// TwinCAT 3 PLC project PLC
// ProgramVersion: 3.1.4023.0
// libraries:
//   Tc2_ControllerToolbox, * (Beckhoff Automation GmbH)
//   Tc2_EtherCAT, * (Beckhoff Automation GmbH)
//   Tc2_Math, * (Beckhoff Automation GmbH)
//   Tc2_ModbusRTU, * (Beckhoff Automation GmbH)
//   Tc2_SerialCom, * (Beckhoff Automation GmbH)
//   Tc2_Standard, * (Beckhoff Automation GmbH)
//   Tc2_System, * (Beckhoff Automation GmbH)
//   Tc2_Utilities, * (Beckhoff Automation GmbH)
//   Tc2_XmlDataSrv, * (Beckhoff Automation GmbH)
//   Tc3_EventLogger, * (Beckhoff Automation GmbH)
//   Tc3_Module, * (Beckhoff Automation GmbH)
// project tree:
//   / MAIN.TcPOU, PlcTask.TcTTO, SerialComTask.TcTTO
//   PMShared/Hardware/Common/Enum/CoE/ EBaudrate.TcDUT, EDataFrame.TcDUT
//   PMShared/Hardware/Common/Enum/ DeviceFamily.TcDUT, DeviceLogLevel.TcDUT, SerialFlowControl.TcDUT, SerialParity.TcDUT
//   PMShared/Hardware/Common/ HardwareManager.TcPOU
//   PMShared/Hardware/Common/Struct/Configs/ AppConfig.TcDUT, DeviceConfiguration.TcDUT, SerialCommunication.TcDUT
//   PMShared/Hardware/Common/Struct/Configs/Calibrate/ CalibrateConfig.TcDUT, CalibratePMsConfig.TcDUT, HSPowermeter.TcDUT, HTPowermeter.TcDUT
//   PMShared/Hardware/Common/Struct/Configs/CanOverEthercat/ CanOverEthercat.TcDUT, CanOverEthercatConfig.TcDUT
//   PMShared/Hardware/Common/Struct/Configs/CanOverEthercat/CoEModules/ CoeSerialComSettings.TcDUT
//   PMShared/Hardware/Common/Struct/Configs/CanOverEthercat/CoEModules/SubModules/ BaudRate.TcDUT, DataFrame.TcDUT, EnableRtsCts.TcDUT, EnableXonXoffRx.TcDUT, EnableXonXoffTx.TcDUT, SubIndexModuleBase.TcDUT
//   PMShared/Hardware/Common/Struct/Configs/Devices/Chuck/WaferPresenceSensor/ WaferPresenceSensor.TcDUT
//   PMShared/Hardware/Common/Struct/Configs/Devices/Powermeter/Sensor/ PowermeterSensor.TcDUT
//   PMShared/Hardware/Common/Struct/Configs/Log/ LogConfig.TcDUT
//   PMShared/Hardware/Common/Struct/Configs/NetIdManagement/ NetIdManagement.TcDUT
//   PMShared/Hardware/Common/Struct/Configs/PMs/ LightspeedConfig.TcDUT, PhotoLumConfig.TcDUT, NstConfig.TcDUT, ProcessModulesConfig.TcDUT, PsdConfig.TcDUT
//   PMShared/Hardware/Common/Tools/CoeAccess/ CoeAccess.TcPOU
//   PMShared/Hardware/Common/Tools/PWM/ PwmGenerator.TcPOU
//   PMShared/Hardware/Common/Tools/SerialCommunication/ SerialCom.TcPOU
//   PMShared/Hardware/Devices/AttenuationFilters/ AttenuationFilterBase.TcPOU
//   PMShared/Hardware/Devices/AttenuationFilters/Configs/ AttenuationFilterConfigs.TcDUT, RotatingSwitchConfigs.TcDUT, SliderAttenuationFilterConfigs.TcDUT
//   PMShared/Hardware/Devices/AttenuationFilters/Configs/SerialCommunication/ BkgrdSerialAttenuation.TcPOU, BkgrdSerialSliderAttenuation.TcPOU, BkgrdSerialRotatingSwitch.TcPOU
//   PMShared/Hardware/Devices/AttenuationFilters/Configs/Thorlabs/ELL14K/ EFeedbackMsgAttenuationELL14k.TcDUT, ELL14kAttenuationFilterConfig.TcDUT
//   PMShared/Hardware/Devices/AttenuationFilters/Configs/Thorlabs/ELL18/ EFeedbackMsgAttenuationELL18.TcDUT, ELL18AttenuationFilterConfig.TcDUT
//   PMShared/Hardware/Devices/AttenuationFilters/Configs/Thorlabs/ELL9/ EFeedbackMsgAttenuationELL9.TcDUT, ELL9AttenuationFilterConfig.TcDUT
//   PMShared/Hardware/Devices/AttenuationFilters/Configs/Thorlabs/ELL6/ EFeedbackMsgAttenuationELL6.TcDUT, ELL6AttenuationFilterConfig.TcDUT
//   PMShared/Hardware/Devices/AttenuationFilters/Configs/Thorlabs/FW212C/ EFeedbackMsgAttenuationFW212C.TcDUT, FW212CAttenuationFilterConfig.TcDUT
//   PMShared/Hardware/Devices/AttenuationFilters/Thorlabs/ ELL14KAttenuationFilter.TcPOU, ELL18AttenuationFilter.TcPOU, ELL9AttenuationFilter.TcPOU, ELL6AttenuationFilter.TcPOU, FW212CAttenuationFilter.TcPOU
//   PMShared/Hardware/Devices/Axes/ AxesBase.TcPOU, AxesConst.TcGVL
//   PMShared/Hardware/Devices/Axes/Configs/ AxesConfigs.TcDUT, IoAxisConfig.TcDUT, IoAxisConfig.TcDUT
//   PMShared/Hardware/Devices/Axes/Configs/Owis/ EFeedbackMsgOwisPs10.TcDUT, Ps10OwisAxisConfig.TcDUT
//   PMShared/Hardware/Devices/Axes/Configs/Owis/SerialCommunication/ BkgrdSerialOwisPs10.TcPOU
//   PMShared/Hardware/Devices/Axes/Configs/Stage/ EFeedbackMsgStage.TcDUT, EStagePosition.TcDUT, IoStageAxisConfig.TcDUT, IoStageStruct.TcDUT, EFeedbackMsgStage.TcDUT, EStagePosition.TcDUT, IoStageAxisConfig.TcDUT, IoStageStruct.TcDUT
//   PMShared/Hardware/Devices/Axes/IoAxis/Stage/ IoStageAxis.TcPOU, IoStageAxis.TcPOU
//   PMShared/Hardware/Devices/Axes/Owis/ Ps10Axis.TcPOU
//   PMShared/Hardware/Devices/Chambers/Configs/ EChamberMode.TcDUT, EFeedbackMsgChamberBase.TcDUT, EFeedbackMsgSlitDoor.TcDUT, ESlitDoorPosition.TcDUT, IoChamberBase.TcDUT, ChamberConfigs.TcDUT
//   PMShared/Hardware/Devices/Chambers/Configs/Lightspeed/ IoLightspeed.TcDUT, IoSafetyLS.TcDUT, LightspeedChamberConfig.TcDUT
//   PMShared/Hardware/Devices/Chambers/Configs/PhotoLum/ EFeedbackMsgPhotoLumChamber.TcDUT, IoChamberPhotoLum.TcDUT, PhotoLumChamberConfig.TcDUT
//   PMShared/Hardware/Devices/Chambers/Configs/PSD/ EFeedbackMsgPsdChamber.TcDUT, IoChamberPsd.TcDUT, PsdChamberConfig.TcDUT, SensorId.TcDUT
//   PMShared/Hardware/Devices/Chambers/Lightspeed/ LightspeedChamber.TcPOU
//   PMShared/Hardware/Devices/Chambers/PhotoLum/ PhotoLumChamber.TcPOU
//   PMShared/Hardware/Devices/Chambers/PSD/ PsdChamber.TcPOU
//   PMShared/Hardware/Devices/Chucks/ ChuckBase.TcPOU
//   PMShared/Hardware/Devices/Chucks/Configs/ ChuckConfigs.TcDUT, EFeedbackMsgChuckBase.TcDUT, EMaterialPresence.TcDUT, EWaferSize.TcDUT
//   PMShared/Hardware/Devices/Chucks/Configs/PhotLum/ EFeedbackMsgPhotoLumChuck.TcDUT, IoChuckPhotoLum.TcDUT, PhotoLumChuckConfig.TcDUT
//   PMShared/Hardware/Devices/Chucks/Configs/PSD/ EFeedbackMsgPsdChuck.TcDUT, IoChuckPsd.TcDUT, PsdChuckConfig.TcDUT
//   PMShared/Hardware/Devices/Chucks/PhotoLum/ PhotoLumChuck.TcPOU
//   PMShared/Hardware/Devices/Chucks/PSD/ PsdChuck.TcPOU
//   PMShared/Hardware/Devices/DistanceSensors/Configs/ DistanceSensorConfigs.TcDUT
//   PMShared/Hardware/Devices/DistanceSensors/Configs/MicroEpsilon/ EFeedbackMsgMicroEpsilonDistanceSensor.TcDUT, MicroEpsilonDistanceSensorConfig.TcDUT, IoMicroEpsilonDistanceSensor.TcDUT
//   PMShared/Hardware/Devices/DistanceSensors/ DistanceSensorBase.TcPOU
//   PMShared/Hardware/Devices/DistanceSensors/MicroEpsilon/ MicroEpsilonDistanceSensor.TcPOU
//   PMShared/Hardware/Devices/FastAttenuation/Configs/ FastAttenuationConfigs.TcDUT
//   PMShared/Hardware/Devices/FastAttenuation/Configs/Parallax/ EFeedbackMsgStd900.TcDUT, IoStd900.TcDUT, Std900FastAttenuationConfig.TcDUT
//   PMShared/Hardware/Devices/FastAttenuation/ FastAttenuationBase.TcPOU
//   PMShared/Hardware/Devices/FastAttenuation/Parallax/ Std900FastAttenuation.TcPOU
//   PMShared/Hardware/Devices/Ffus/Astrofan/ Astrofan612Ffu.TcPOU, Constants.TcGVL
//   PMShared/Hardware/Devices/Ffus/Astrofan/Loop/EventRaise/ EventRaised.TcPOU
//   PMShared/Hardware/Devices/Ffus/Astrofan/Loop/FfuSpeedMatrix/ Ffumatrixconfig.TcDUT, FfuSpeed.TcDUT, ScaleSpeed.TcPOU
//   PMShared/Hardware/Devices/Ffus/Configs/Astrofan/ Astrofan612FfuConfig.TcDUT, Astrofan612FfuLoopConfig.TcDUT, Astrofan612FfuEvent.TcDUT, EFeedbackMsgAstrofan612.TcDUT
//   PMShared/Hardware/Devices/Ffus/Configs/ FfuConfigs.TcDUT
//   PMShared/Hardware/Devices/Ffus/ FfuBase.TcPOU
//   PMShared/Hardware/Devices/FiberSwitch/Configs/ FiberSwitchConfigs.TcDUT
//   PMShared/Hardware/Devices/FiberSwitch/Configs/Leoni/ EFeedbackMsgEol.TcDUT, EOLFiberSwitchConfig.TcDUT
//   PMShared/Hardware/Devices/FiberSwitch/Configs/SerialCommunication/ BkgrdSerialFiberSwitch.TcPOU
//   PMShared/Hardware/Devices/FiberSwitch/ FiberSwitchBase.TcPOU
//   PMShared/Hardware/Devices/FiberSwitch/Leoni/ EOLFiberSwitch.TcPOU
//   PMShared/Hardware/Devices/Ionizers/Configs/ IonizerAlarm.TcDUT, IonizerConfigs.TcDUT, IonizerConst.TcGVL
//   PMShared/Hardware/Devices/Ionizers/Configs/Keyence/ EFeedbackMsgSJH108.TcDUT, IoSJH108A.TcDUT, SJH108IonizerConfig.TcDUT
//   PMShared/Hardware/Devices/Ionizers/ IonizerBase.TcPOU
//   PMShared/Hardware/Devices/Ionizers/Keyence/ SJH108Ionizer.TcPOU
//   PMShared/Hardware/Devices/Lasers/Coherent/ Sapphire488Laser.TcPOU
//   PMShared/Hardware/Devices/Lasers/Configs/Base/ HoursStruct.TcDUT
//   PMShared/Hardware/Devices/Lasers/Configs/Coherent/ EFeedbackMsgSapphire488.TcDUT, Sapphire488LaserConfig.TcDUT
//   PMShared/Hardware/Devices/Lasers/Configs/ LaserConfigs.TcDUT
//   PMShared/Hardware/Devices/Lasers/Configs/Leukos/ EControlModePiano450.TcDUT, EFeedbackMsgPiano450.TcDUT, Piano450LaserConfig.TcDUT
//   PMShared/Hardware/Devices/Lasers/Configs/Quantum/ EControlModeSmd12.TcDUT, EFeedbackMsgSMD12.TcDUT, SMD12LaserConfig.TcDUT
//   PMShared/Hardware/Devices/Lasers/Configs/SerialCommunication/ BkgrdSerialLaser.TcPOU
//   PMShared/Hardware/Devices/Lasers/ LaserBase.TcPOU
//   PMShared/Hardware/Devices/Lasers/Leukos/ Piano450Laser.TcPOU
//   PMShared/Hardware/Devices/Lasers/Quantum/ SMD12Laser.TcPOU
//   PMShared/Hardware/Devices/Lights/Arduino/ ArduinoLight.TcPOU
//   PMShared/Hardware/Devices/Lights/Configs/Evosens/ EvosensLightConfig.TcDUT, EFeedbackMsgEvosensLight.TcDUT
//   PMShared/Hardware/Devices/Lights/Configs/Arduino/ EFeedbackMsgArduinoLight.TcDUT, ArduinoLightConfig.TcDUT
//   PMShared/Hardware/Devices/Lights/Configs/ LightConfigs.TcDUT
//   PMShared/Hardware/Devices/Lights/Configs/SerialCommunication/ BkgrdSerialLight.TcPOU
//   PMShared/Hardware/Devices/Lights/Evosens/ EvosensLight.TcPOU
//   PMShared/Hardware/Devices/Lights/ LightBase.TcPOU
//   PMShared/Hardware/Devices/MPPCs/Configs/Hamamatsu/ C13336MppcConfig.TcDUT, EFeedbackMsgC13336.TcDUT, EMppcCollector.TcDUT, EMppcStateModule.TcDUT, IoC13336Mppc.TcDUT
//   PMShared/Hardware/Devices/MPPCs/Configs/ MppcConfigs.TcDUT
//   PMShared/Hardware/Devices/MPPCs/Configs/SerialCommunication/ BkgrdSerialMppcNarrow.TcPOU, BkgrdSerialMppcWide.TcPOU
//   PMShared/Hardware/Devices/MPPCs/Hamamatsu/C13336/ C13336MppcWide.TcPOU, C13366MppcNarrow.TcPOU
//   PMShared/Hardware/Devices/MPPCs/Hamamatsu/ C13336Mppc.TcPOU
//   PMShared/Hardware/Devices/MPPCs/ MppcBase.TcPOU
//   PMShared/Hardware/Devices/OpticalPowermeters/Configs/ OpticalPowermeterConfigs.TcDUT
//   PMShared/Hardware/Devices/OpticalPowermeters/Configs/SerialCommunication/ BkgrdSerialOpticalPowermeterHs.TcPOU, BkgrdSerialOpticalPowermeterHt.TcPOU
//   PMShared/Hardware/Devices/OpticalPowermeters/Configs/Thorlabs/ EFeedbackMsgPM101.TcDUT, EPowerIlluminationFlow.TcDUT, IoControlPM101.TcDUT, PM101OpticalPowermeterConfig.TcDUT
//   PMShared/Hardware/Devices/OpticalPowermeters/ OpticalPowermeterBase.TcPOU
//   PMShared/Hardware/Devices/OpticalPowermeters/Thorlabs/PM101/Messages/ BeamDiameterMsg.TcDUT, AttenuationMsg.TcDUT, SensorTypeMsg.TcDUT, ResponsivityMsg.TcDUT, CustomMsg.TcDUT, IdentifierMsg.TcDUT, MaxPowerMsg.TcDUT, MinPowerMsg.TcDUT, PowerMsg.TcDUT, WavelengthMsg.TcDUT, WavelengthRangeMsg.TcDUT
//   PMShared/Hardware/Devices/OpticalPowermeters/Thorlabs/PM101/ PM101OpticalPowermeterHs.TcPOU, PM101OpticalPowermeterHt.TcPOU
//   PMShared/Hardware/Devices/OpticalPowermeters/Thorlabs/ PM101OpticalPowermeter.TcPOU
//   PMShared/Hardware/Devices/PolarisationFilters/Configs/ PolarisationFilterConfigs.TcDUT
//   PMShared/Hardware/Devices/PolarisationFilters/Configs/SerialCommunication/ BkgrdSerialPolarisation.TcPOU
//   PMShared/Hardware/Devices/PolarisationFilters/Configs/Thorlabs/ELL14K/ EFeedbackMsgPolarisationELL14K.TcDUT, ELL14KPolarisationFilterConfig.TcDUT
//   PMShared/Hardware/Devices/PolarisationFilters/Configs/Thorlabs/ EPolar.TcDUT
//   PMShared/Hardware/Devices/PolarisationFilters/Configs/Thorlabs/FW212C/ EFeedbackMsgPolarisationFW212C.TcDUT, FW212CPolarisationFilterConfig.TcDUT
//   PMShared/Hardware/Devices/PolarisationFilters/ PolarisationFilterBase.TcPOU
//   PMShared/Hardware/Devices/PolarisationFilters/Thorlabs/ ELL14KPolarisationFilter.TcPOU, FW212CPolarisationFilter.TcPOU
//   PMShared/Hardware/Devices/Chambers/ ChamberBase.TcPOU
//   PMShared/Hardware/Devices/Rfids/Balluff/ BisL405Rfid.TcPOU
//   PMShared/Hardware/Devices/Rfids/Configs/Balluff/ BisL405RfidConfig.TcDUT, EFeedbackMsgBisL405.TcDUT, IoBisL405Rfid.TcDUT
//   PMShared/Hardware/Devices/Rfids/Configs/ RfidConfigs.TcDUT
//   PMShared/Hardware/Devices/Rfids/ RfidBase.TcPOU
//   PMShared/Hardware/Devices/Safety/Configs/ Interlock.TcDUT
//   PMShared/Hardware/Devices/Safety/ Safety.TcPOU
//   PMShared/Hardware/Devices/Screens/Configs/Densitron/ DM430GNScreenConfig.TcDUT, EDisplayControlStep.TcDUT, EFeedbackMsgDM430GN.TcDUT, EScreenSide.TcDUT
//   PMShared/Hardware/Devices/Screens/Configs/ ScreenConfigs.TcDUT
//   PMShared/Hardware/Devices/Screens/Configs/SerialCommunication/ BkgrdSerialScreenFS.TcPOU, BkgrdSerialScreenBS.TcPOU
//   PMShared/Hardware/Devices/Screens/Densitron/ DM430GNScreen.TcPOU
//   PMShared/Hardware/Devices/Screens/Densitron/DM430GNS/ DM430GNScreenBS.TcPOU, DM430GNScreenFS.TcPOU
//   PMShared/Hardware/Devices/Screens/ ScreenBase.TcPOU
//   PMShared/Hardware/Devices/Shutters/Configs/Eopc/ Sh10pilShutterConfig.TcDUT, EFeedbackMsgSh10pil.TcDUT, IoSh10pilShutter.TcDUT
//   PMShared/Hardware/Devices/Shutters/Configs/ ShutterConfigs.TcDUT
//   PMShared/Hardware/Devices/Shutters/Configs/Uniblitz/ Ed12dssShutterConfig.TcDUT, EFeedbackMsgEd12dss.TcDUT, IoEd12dssShutter.TcDUT
//   PMShared/Hardware/Devices/Shutters/Eopc/ Sh10pilShutter.TcPOU
//   PMShared/Hardware/Devices/Shutters/ ShutterBase.TcPOU
//   PMShared/Hardware/Devices/Shutters/Uniblitz/ Ed12dssShutter.TcPOU
//   PMShared/Hardware/Interface/ IDevice.TcIO
//   PMShared/Hardware/Interface/TrackExecution/ IExecution.TcIO, TExecution.TcPOU, TExecutionState.TcDUT
//   Service/PMs/ EFeedbackMsgPlc.TcDUT, PlcModule.TcPOU
//   Service/PMs/Lightspeed/Calibrate/ LsCalibrateConfig.TcDUT, PolarisationConfig.TcDUT, ResponsivityConfig.TcDUT, RFactorBase.TcDUT, RFactorSettings.TcDUT
//   Service/PMs/Lightspeed/Communication/RS232/ LsBkgrdLsSerialCom.TcPOU
//   Service/PMs/Lightspeed/ Lightspeed.TcPOU
//   Service/PMs/Nst/Communication/RS232/ NstBkgrdLsSerialCom.TcPOU
//   Service/PMs/Nst/ Nst.TcPOU
//   Service/PMs/PhotoLum/Communication/RS232/ PhotoLumBkgrdSerialCom.TcPOU
//   Service/PMs/PhotoLum/ PhotoLum.TcPOU
//   Service/PMs/Psd/Communication/RS232/ PsdBkgrdSerialCom.TcPOU
//   Service/PMs/Psd/ Psd.TcPOU
//   Shared/GlobalVariables/ Const.TcGVL, GlobalConfig.TcGVL, HardwareGlobalVariables.TcGVL
//   Shared/Log/ ILogger.TcIO, LogEventLevel.TcDUT, Logger.TcPOU
//   Shared/Tools/StringBuilder/ ILimitedStringBuilder.TcIO, IStringBuilder.TcIO, StringBuilder.TcPOU
//   Shared/Tools/Trigger/ Trigger.TcPOU
//   Shared/Tools/Xml/ TXml.TcPOU
//   Service/ HardwareControl.TcPOU
// real-time tasks:
//   TASK PlcTask: cycle T#10ms, priority 20, ADS port 350
//   TASK SerialComTask: cycle T#10ms, priority 2, ADS port 351
// I/O:
//   DEVICE Device 1 (EtherCAT), AmsNetId 5.108.191.186.2.1
//     Term 1 (EK1200) [EK1200-5000 EtherCAT Power supply (2A E-Bus)]
//       Term 2 (EK1122) [EK1122 2 port EtherCAT junction]
//       Term 3 (EL6002) [EL6002 Interface 2Ch. (RS232)]
//       Term 4 (EK1110) [EK1110 EtherCAT extension]
// variable links:
//   PLC/PLC Instance <-> Device 1 (EtherCAT)/Term 1 (EK1200)/Term 3 (EL6002)
//     SerialComTask Inputs/BkgrdSerialOwisPs10.stInFilterWheel @bit {16..184 step 8} <-> COM TxPDO-Map Inputs Channel 1/Data In {0..21}  (22 links)
//     SerialComTask Inputs/BkgrdSerialOwisPs10.stInFilterWheel <-> COM TxPDO-Map Inputs Channel 1/Status
//     SerialComTask Outputs/BkgrdSerialOwisPs10.stOutFilterWheel <-> COM RxPDO-Map Outputs Channel 1/Ctrl
//     SerialComTask Outputs/BkgrdSerialOwisPs10.stOutFilterWheel @bit {16..184 step 8} <-> COM RxPDO-Map Outputs Channel 1/Data Out {0..21}  (22 links)

CONFIGURATION PLC
    RESOURCE PLC ON TwinCAT3
        TASK PlcTask(INTERVAL := T#10ms, PRIORITY := 20);
        TASK SerialComTask(INTERVAL := T#10ms, PRIORITY := 2);
        PROGRAM MAIN WITH PlcTask : MAIN;
        PROGRAM LsBkgrdLsSerialCom WITH SerialComTask : LsBkgrdLsSerialCom;
        PROGRAM NstBkgrdLsSerialCom WITH SerialComTask : NstBkgrdLsSerialCom;
        PROGRAM PhotoLumBkgrdSerialCom WITH SerialComTask : PhotoLumBkgrdSerialCom;
        PROGRAM PsdBkgrdSerialCom WITH SerialComTask : PsdBkgrdSerialCom;
    END_RESOURCE
END_CONFIGURATION

// ---- PMShared/Hardware/Common/Enum/CoE/EBaudrate.TcDUT
{attribute 'qualified_only'}
{attribute 'strict'}
{attribute 'to_string'}
TYPE EBaudrate :
(
	_9600   := 6,
	_19200  := 7,
	_38400  := 8,
	_57600  := 9,
	_115200 := 10
);
END_TYPE

// ---- PMShared/Hardware/Common/Enum/CoE/EDataFrame.TcDUT
{attribute 'qualified_only'}
{attribute 'strict'}
{attribute 'to_string'}
TYPE EDataFrame :
(
	_8N1 := 3,
	_8E1 := 4
);
END_TYPE

// ---- PMShared/Hardware/Common/Enum/DeviceFamily.TcDUT
{attribute 'qualified_only'}
{attribute 'strict'}
{attribute 'to_string'}
TYPE DeviceFamily :
(	
	Other := -1,
	Chamber := 0,
	AttenuationFilter,
	Chuck,
	DistanceSensors,
	FiberSwitch,
	Laser,
	MotionControl,
	MPPC,
	OpticalPowermeter,
	PolarisationFilter,
	Shutter,
	FastAttenuation,
	Axes,
	Light,
	Screen,
	Ffu,
	Rfid,
	Ionizer
);
END_TYPE

// ---- PMShared/Hardware/Common/Enum/DeviceLogLevel.TcDUT
{attribute 'qualified_only'}
{attribute 'strict'}
TYPE DeviceLogLevel :
(
	None := 0,
    Verbose,
    Debug,
    Information,
    Warning,
    Error
);
END_TYPE

// ---- PMShared/Hardware/Common/Enum/SerialFlowControl.TcDUT
{attribute 'qualified_only'}
{attribute 'strict'}
{attribute 'to_string'}
TYPE SerialFlowControl :
(
	None := 0,
	XonXoff,
	RtsCts,
	DsrDts
);
END_TYPE

// ---- PMShared/Hardware/Common/Enum/SerialParity.TcDUT
{attribute 'qualified_only'}
{attribute 'strict'}
TYPE SerialParity :
(
	None := 0,
	Odd,
	Even,
	Mark,
	Space
);
END_TYPE

// ---- PMShared/Hardware/Common/Struct/Configs/AppConfig.TcDUT
TYPE AppConfig :
STRUCT
	NetIdManagement : NetIdManagement;
	CanOverEthercatConfig : CanOverEthercatConfig;
	LogConfig : LogConfig;
	CalibrateConfig : CalibrateConfig;
END_STRUCT
END_TYPE

// ---- PMShared/Hardware/Common/Struct/Configs/Calibrate/CalibrateConfig.TcDUT
TYPE CalibrateConfig :
STRUCT
	CalibratePath : STRING;
	CalibrateHeaderNodeXml : STRING;
END_STRUCT
END_TYPE

// ---- PMShared/Hardware/Common/Struct/Configs/Calibrate/CalibratePMsConfig.TcDUT
{attribute 'OPC.UA.DA' := '0'}
TYPE CalibratePMsConfig :
STRUCT
	LsCalibrateConfig : LsCalibrateConfig;
END_STRUCT
END_TYPE

// ---- PMShared/Hardware/Common/Struct/Configs/Calibrate/HSPowermeter.TcDUT
{attribute 'OPC.UA.DA' := '0'}
TYPE HSPowermeter :
STRUCT
	PolarisationConfig : PolarisationConfig;
	RFactorSettings : RFactorSettings;
	ResponsivityConfig : ResponsivityConfig;
END_STRUCT
END_TYPE

// ---- PMShared/Hardware/Common/Struct/Configs/Calibrate/HTPowermeter.TcDUT
{attribute 'OPC.UA.DA' := '0'}
TYPE HTPowermeter :
STRUCT
	PolarisationConfig : PolarisationConfig;
	RFactorSettings : RFactorSettings;
	ResponsivityConfig : ResponsivityConfig;
END_STRUCT
END_TYPE

// ---- PMShared/Hardware/Common/Struct/Configs/CanOverEthercat/CanOverEthercat.TcDUT
{attribute 'OPC.UA.DA' := '0'}
TYPE CanOverEthercat :
STRUCT
	AdrEthercat : UINT;
END_STRUCT
END_TYPE

// ---- PMShared/Hardware/Common/Struct/Configs/CanOverEthercat/CanOverEthercatConfig.TcDUT
TYPE CanOverEthercatConfig :
STRUCT
	CoeSerialComSettings : CoeSerialComSettings;
END_STRUCT
END_TYPE

// ---- PMShared/Hardware/Common/Struct/Configs/CanOverEthercat/CoEModules/CoeSerialComSettings.TcDUT
TYPE CoeSerialComSettings :
STRUCT
	IndexComPort1 : STRING;
	IndexComPort2 : STRING;
	EnableRtsCts : EnableRtsCts;
	EnableXonXoffTx : EnableXonXoffTx;
	EnableXonXoffRx : EnableXonXoffRx;
	BaudRate : BaudRate;
	DataFrame : DataFrame;
END_STRUCT
END_TYPE

// ---- PMShared/Hardware/Common/Struct/Configs/CanOverEthercat/CoEModules/SubModules/BaudRate.TcDUT
TYPE BaudRate EXTENDS SubIndexModuleBase :
STRUCT
END_STRUCT
END_TYPE

// ---- PMShared/Hardware/Common/Struct/Configs/CanOverEthercat/CoEModules/SubModules/DataFrame.TcDUT
TYPE DataFrame EXTENDS SubIndexModuleBase :
STRUCT
END_STRUCT
END_TYPE

// ---- PMShared/Hardware/Common/Struct/Configs/CanOverEthercat/CoEModules/SubModules/EnableRtsCts.TcDUT
TYPE EnableRtsCts EXTENDS SubIndexModuleBase :
STRUCT
END_STRUCT
END_TYPE

// ---- PMShared/Hardware/Common/Struct/Configs/CanOverEthercat/CoEModules/SubModules/EnableXonXoffRx.TcDUT
TYPE EnableXonXoffRx EXTENDS SubIndexModuleBase :
STRUCT
END_STRUCT
END_TYPE

// ---- PMShared/Hardware/Common/Struct/Configs/CanOverEthercat/CoEModules/SubModules/EnableXonXoffTx.TcDUT
TYPE EnableXonXoffTx EXTENDS SubIndexModuleBase :
STRUCT
END_STRUCT
END_TYPE

// ---- PMShared/Hardware/Common/Struct/Configs/CanOverEthercat/CoEModules/SubModules/SubIndexModuleBase.TcDUT
TYPE SubIndexModuleBase :
STRUCT
	SubIndex : STRING;
	SizeByte  : UDINT;
END_STRUCT
END_TYPE

// ---- PMShared/Hardware/Common/Struct/Configs/DeviceConfiguration.TcDUT
TYPE DeviceConfiguration :
STRUCT
	{attribute 'OPC.UA.DA' := '0'}
	Name : STRING;
	{attribute 'OPC.UA.DA' := '1'}
	DeviceID : STRING;	
	{attribute 'OPC.UA.DA' := '1'}
	IsEnabled : BOOL;
	{attribute 'OPC.UA.DA' := '0'}
	IsSimulated : BOOL;
	{attribute 'OPC.UA.DA' := '0'}
	LogLevel : DeviceLogLevel := DeviceLogLevel.Debug;
END_STRUCT
END_TYPE

// ---- PMShared/Hardware/Common/Struct/Configs/Devices/Chuck/WaferPresenceSensor/WaferPresenceSensor.TcDUT
{attribute 'OPC.UA.DA' := '0'}
TYPE WaferPresenceSensor :
STRUCT
	Name : STRING;
	Diameter : UINT;
	InputWaferPresence AT %I* : BOOL;
END_STRUCT
END_TYPE

// ---- PMShared/Hardware/Common/Struct/Configs/Devices/Powermeter/Sensor/PowermeterSensor.TcDUT
{attribute 'OPC.UA.DA' := '0'}
TYPE PowermeterSensor :
STRUCT
	Name : STRING;
	Wavelength : UINT;
	Attenuation : UINT;
END_STRUCT
END_TYPE

// ---- PMShared/Hardware/Common/Struct/Configs/Log/LogConfig.TcDUT
TYPE LogConfig :
STRUCT
	LogFileConfigPath : STRING;
	HeaderNodeXml : STRING;
	LogFilePath : STRING;
	AddLogsConsole : BOOL;
END_STRUCT
END_TYPE

// ---- PMShared/Hardware/Common/Struct/Configs/NetIdManagement/NetIdManagement.TcDUT
TYPE NetIdManagement :
STRUCT
	TargetNetId : STRING;
	FirstPeripheral : STRING;
END_STRUCT
END_TYPE

// ---- PMShared/Hardware/Common/Struct/Configs/PMs/LightspeedConfig.TcDUT
TYPE LightspeedConfig :
STRUCT
	DeviceID : STRING;
	IsEnabled : BOOL;
	Version : STRING;
	ChamberConfigs : ChamberConfigs;	
	AttenuationFilterConfigs : AttenuationFilterConfigs;
	PolarisationFilterConfigs : PolarisationFilterConfigs;
	SliderAttenuationFilterConfigs : SliderAttenuationFilterConfigs;
	RotatingSwitchConfigs : RotatingSwitchConfigs;
	LaserConfigs : LaserConfigs;
	FiberSwitchConfigs : FiberSwitchConfigs;
	OpticalPowermeterConfigs : OpticalPowermeterConfigs;
	DistanceSensorConfigs : DistanceSensorConfigs;
	MppcConfigs : MppcConfigs;
	ShutterConfigs : ShutterConfigs; 
	FastAttenuationConfigs : FastAttenuationConfigs;
END_STRUCT
END_TYPE

// ---- PMShared/Hardware/Common/Struct/Configs/PMs/PhotoLumConfig.TcDUT
TYPE PhotoLumConfig :
STRUCT
	DeviceID : STRING;
	IsEnabled : BOOL;
	SafetyIsEnabled : BOOL;
	ChamberConfigs : ChamberConfigs;
	ChuckConfigs : ChuckConfigs;	
	AxesConfigs : AxesConfigs;
	LightConfigs : LightConfigs;
	DistanceSensorConfigs : DistanceSensorConfigs;
END_STRUCT
END_TYPE

// ---- PMShared/Hardware/Common/Struct/Configs/PMs/NstConfig.TcDUT
TYPE NstConfig :
STRUCT
	DeviceID : STRING;
	IsEnabled : BOOL;
	AttenuationFilterConfigs : AttenuationFilterConfigs;
	LaserConfigs : LaserConfigs;
	ShutterConfigs : ShutterConfigs; 
	FastAttenuationConfigs : FastAttenuationConfigs;
	IonizerConfigs 	: IonizerConfigs; 
	FfuConfigs 		: FfuConfigs;	
END_STRUCT
END_TYPE

// ---- PMShared/Hardware/Common/Struct/Configs/PMs/ProcessModulesConfig.TcDUT
TYPE ProcessModulesConfig :
STRUCT
	PsdConfig : PsdConfig;
	LightspeedConfig : LightspeedConfig;	
	NstConfig : NstConfig;
	PhotoLumConfig : PhotoLumConfig;
END_STRUCT
END_TYPE

// ---- PMShared/Hardware/Common/Struct/Configs/PMs/PsdConfig.TcDUT
TYPE PsdConfig :
STRUCT
	DeviceID : STRING;
	IsEnabled : BOOL;
	SafetyIsEnabled : BOOL;
	ChamberConfigs : ChamberConfigs;
	AxesConfigs : AxesConfigs;	
	ChuckConfigs : ChuckConfigs;
	ScreenConfigs : ScreenConfigs;
	FfuConfigs : FfuConfigs;
	RfidConfigs : RfidConfigs;
END_STRUCT
END_TYPE

// ---- PMShared/Hardware/Common/Struct/Configs/SerialCommunication.TcDUT
{attribute 'OPC.UA.DA' := '0'}
TYPE SerialCommunication :
STRUCT
	Port : STRING;
	BaudRate : UDINT;
	DataFrame : STRING;
	FlowControl : SerialFlowControl;
	CanOverEthercat : CanOverEthercat;
END_STRUCT
END_TYPE

// ---- PMShared/Hardware/Devices/AttenuationFilters/Configs/AttenuationFilterConfigs.TcDUT
TYPE AttenuationFilterConfigs :
STRUCT
	FW212CAttenuationFilterConfig : FW212CAttenuationFilterConfig;
	ELL14KAttenuationFilterConfig : ELL14KAttenuationFilterConfig;
	ELL18AttenuationFilterConfig : ELL18AttenuationFilterConfig;
	ELL9AttenuationFilterConfig : ELL9AttenuationFilterConfig;
	ELL6AttenuationFilterConfig : ELL6AttenuationFilterConfig;
END_STRUCT
END_TYPE

// ---- PMShared/Hardware/Devices/AttenuationFilters/Configs/RotatingSwitchConfigs.TcDUT
TYPE RotatingSwitchConfigs :
STRUCT
	ELL18RotatingSwitchConfig : ELL18AttenuationFilterConfig;
END_STRUCT
END_TYPE

// ---- PMShared/Hardware/Devices/AttenuationFilters/Configs/SliderAttenuationFilterConfigs.TcDUT
TYPE SliderAttenuationFilterConfigs :
STRUCT
	ELL6SliderFilterConfig : ELL6AttenuationFilterConfig;
END_STRUCT
END_TYPE

// ---- PMShared/Hardware/Devices/AttenuationFilters/Configs/Thorlabs/ELL14K/EFeedbackMsgAttenuationELL14k.TcDUT
{attribute 'qualified_only'}
{attribute 'strict'}
TYPE EFeedbackMsgAttenuationELL14k :
(
	StateMsg := 1,
	PositionMsg := 10,
    IdMsg,
    CustomMsg
);
END_TYPE

// ---- PMShared/Hardware/Devices/AttenuationFilters/Configs/Thorlabs/ELL14K/ELL14kAttenuationFilterConfig.TcDUT
TYPE ELL14kAttenuationFilterConfig EXTENDS DeviceConfiguration :
STRUCT
	SerialCommunication : SerialCommunication;
END_STRUCT
END_TYPE

// ---- PMShared/Hardware/Devices/AttenuationFilters/Configs/Thorlabs/ELL18/EFeedbackMsgAttenuationELL18.TcDUT
{attribute 'qualified_only'}
{attribute 'strict'}
TYPE EFeedbackMsgAttenuationELL18 :
(
	StateMsg := 1,
	PositionMsg := 10,
    IdMsg,
    CustomMsg
);
END_TYPE

// ---- PMShared/Hardware/Devices/AttenuationFilters/Configs/Thorlabs/ELL18/ELL18AttenuationFilterConfig.TcDUT
TYPE ELL18AttenuationFilterConfig EXTENDS DeviceConfiguration :
STRUCT
	SerialCommunication : SerialCommunication;
END_STRUCT
END_TYPE

// ---- PMShared/Hardware/Devices/AttenuationFilters/Configs/Thorlabs/ELL9/EFeedbackMsgAttenuationELL9.TcDUT
{attribute 'qualified_only'}
{attribute 'strict'}
TYPE EFeedbackMsgAttenuationELL9 :
(
	StateMsg := 1,
	StatusMsg := 2,
	IsAliveMsg := 3,
	PositionMsg := 10,	
    IdMsg,
    CustomMsg	
);
END_TYPE

// ---- PMShared/Hardware/Devices/AttenuationFilters/Configs/Thorlabs/ELL9/ELL9AttenuationFilterConfig.TcDUT
TYPE ELL9AttenuationFilterConfig EXTENDS DeviceConfiguration :
STRUCT
	SerialCommunication : SerialCommunication;
END_STRUCT
END_TYPE

// ---- PMShared/Hardware/Devices/AttenuationFilters/Configs/Thorlabs/ELL6/EFeedbackMsgAttenuationELL6.TcDUT
{attribute 'qualified_only'}
{attribute 'strict'}
TYPE EFeedbackMsgAttenuationELL6 :
(
	StateMsg := 1,
	PositionMsg := 10,
    IdMsg,
    CustomMsg	
);
END_TYPE

// ---- PMShared/Hardware/Devices/AttenuationFilters/Configs/Thorlabs/ELL6/ELL6AttenuationFilterConfig.TcDUT
TYPE ELL6AttenuationFilterConfig EXTENDS DeviceConfiguration :
STRUCT
	SerialCommunication : SerialCommunication;
END_STRUCT
END_TYPE

// ---- PMShared/Hardware/Devices/AttenuationFilters/Configs/Thorlabs/FW212C/EFeedbackMsgAttenuationFW212C.TcDUT
{attribute 'qualified_only'}
{attribute 'strict'}
TYPE EFeedbackMsgAttenuationFW212C :
(
	CheckConnectionMsg := 10,
    PositionMsg,
    PositionCountMsg,
    IdMsg,
    CustomMsg
);
END_TYPE

// ---- PMShared/Hardware/Devices/AttenuationFilters/Configs/Thorlabs/FW212C/FW212CAttenuationFilterConfig.TcDUT
TYPE FW212CAttenuationFilterConfig EXTENDS DeviceConfiguration :
STRUCT
	SerialCommunication : SerialCommunication;
END_STRUCT
END_TYPE

// ---- PMShared/Hardware/Devices/Axes/Configs/AxesConfigs.TcDUT
TYPE AxesConfigs :
STRUCT
	IoStageAxisConfig : IoStageAxisConfig;	
	Ps10OwisAxisConfig : Ps10OwisAxisConfig;
END_STRUCT
END_TYPE

// ---- PMShared/Hardware/Devices/Axes/Configs/IoAxisConfig.TcDUT
TYPE IoAxisConfig EXTENDS DeviceConfiguration :
STRUCT
END_STRUCT
END_TYPE

// ---- PMShared/Hardware/Devices/Axes/Configs/Owis/EFeedbackMsgOwisPs10.TcDUT
{attribute 'qualified_only'}
{attribute 'strict'}
TYPE EFeedbackMsgOwisPs10 :
(
	StateMsg := 1,
	AxisStateMsg := 2,
	IsAliveMsg := 3,
	DrivingCurrentMsg := 10,
	HoldingCurrentMsg,	
	LimitSwitchMsg,
	ErrMsg,
	PositionMsg := 20,	
	IsInMovingMsg,	
	CurrentPositionCounterMsg,
	CustomMsg := 50	
);
END_TYPE

// ---- PMShared/Hardware/Devices/Axes/Configs/Owis/Ps10OwisAxisConfig.TcDUT
TYPE Ps10OwisAxisConfig EXTENDS DeviceConfiguration :
STRUCT
	SerialCommunication : SerialCommunication;
END_STRUCT
END_TYPE

// ---- PMShared/Hardware/Devices/Axes/Configs/Stage/EFeedbackMsgStage.TcDUT
{attribute 'strict'}
TYPE EFeedbackMsgStage :
(
	PositionMsg := 10
);
END_TYPE

// ---- PMShared/Hardware/Devices/Axes/Configs/Stage/EStagePosition.TcDUT
{attribute 'qualified_only'}
{attribute 'strict'}
TYPE EStagePosition :
(
	Unknown := 0,
	Loading,
	Process
);
END_TYPE

// ---- PMShared/Hardware/Devices/Axes/Configs/Stage/IoStageAxisConfig.TcDUT
TYPE IoStageAxisConfig EXTENDS IoAxisConfig :
STRUCT
END_STRUCT
END_TYPE

// ---- PMShared/Hardware/Devices/Axes/Configs/Stage/IoStageStruct.TcDUT
TYPE IoStageStruct :
STRUCT
    InputLoadingPosition AT %I* : INT;
    InputProcessPosition AT %I* : INT;	
	
	OutputLoadingPosition AT %Q* : BOOL;
	OutputProcessPosition AT %Q* : BOOL;			
END_STRUCT
END_TYPE

// ---- PMShared/Hardware/Devices/Axes/Configs/IoAxisConfig.TcDUT
TYPE IoAxisConfig EXTENDS DeviceConfiguration :
STRUCT
END_STRUCT
END_TYPE

// ---- PMShared/Hardware/Devices/Axes/Configs/Stage/EFeedbackMsgStage.TcDUT
{attribute 'strict'}
TYPE EFeedbackMsgStage :
(
	PositionMsg := 10
);
END_TYPE

// ---- PMShared/Hardware/Devices/Axes/Configs/Stage/EStagePosition.TcDUT
{attribute 'qualified_only'}
{attribute 'strict'}
TYPE EStagePosition :
(
	Unknown := 0,
	Loading,
	Process
);
END_TYPE

// ---- PMShared/Hardware/Devices/Axes/Configs/Stage/IoStageAxisConfig.TcDUT
TYPE IoStageAxisConfig EXTENDS IoAxisConfig :
STRUCT
END_STRUCT
END_TYPE

// ---- PMShared/Hardware/Devices/Axes/Configs/Stage/IoStageStruct.TcDUT
TYPE IoStageStruct :
STRUCT
    InputLoadingPosition AT %I* : INT;
    InputProcessPosition AT %I* : INT;	
	
	OutputLoadingPosition AT %Q* : BOOL;
	OutputProcessPosition AT %Q* : BOOL;			
END_STRUCT
END_TYPE

// ---- PMShared/Hardware/Devices/Chambers/Configs/EChamberMode.TcDUT
{attribute 'qualified_only'}
{attribute 'strict'}
TYPE EChamberMode :
(
	Unknown := 0,
	Maintenance,
	Run
);
END_TYPE

// ---- PMShared/Hardware/Devices/Chambers/Configs/EFeedbackMsgChamberBase.TcDUT
{attribute 'qualified_only'}
{attribute 'strict'}
TYPE EFeedbackMsgChamberBase :
(
	IsInMaintenanceMsg := 10,
	ArmNotExtendedMsg,
	EfemSlitDoorOpenPositionMsg,
	IsReadyToLoadUnloadMsg
);
END_TYPE

// ---- PMShared/Hardware/Devices/Chambers/Configs/EFeedbackMsgSlitDoor.TcDUT
{attribute 'strict'}
TYPE EFeedbackMsgSlitDoor :
(
	PositionMsg := 10
);
END_TYPE

// ---- PMShared/Hardware/Devices/Chambers/Configs/ESlitDoorPosition.TcDUT
{attribute 'qualified_only'}
{attribute 'strict'}
TYPE ESlitDoorPosition :
(
	Unknown := 0,
	Open,
	Close,
	Error
);
END_TYPE

// ---- PMShared/Hardware/Devices/Chambers/Configs/IoChamberBase.TcDUT
{attribute 'OPC.UA.DA' := '1'}
TYPE IoChamberBase :
STRUCT
	(** Physical inputs **)	
		
	{attribute 'OPC.UA.DA.Access' := '1'}
    InputIsInMaintenance	AT %I* : BOOL;		
	{attribute 'OPC.UA.DA.Access' := '1'}
    InputArmNotExtended		AT %I* : BOOL;
	
	{attribute 'OPC.UA.DA.Access' := '1'}
	InputEfemSlitDoorOpen AT %I* : BOOL;		
	OutputIsReadyToLoadUnload AT %Q* : BOOL;		
END_STRUCT
END_TYPE

// ---- PMShared/Hardware/Devices/Chambers/Configs/Lightspeed/IoLightspeed.TcDUT
{attribute 'OPC.UA.DA' := '1'}
TYPE IoLightspeed EXTENDS IoChamberBase :
STRUCT
	(** Physical inputs **)	
	
	(** ON input : **)
	(** OFF input :  **)
	(** Default :  **)
	{attribute 'OPC.UA.DA.Access' := '1'}
    InputIsWaferPresence	AT %I* : BOOL;
	
	{attribute 'OPC.UA.DA.Access' := '1'}
    InputAdvancedUserMode	AT %I* : BOOL;
	
	{attribute 'OPC.UA.DA.Access' := '1'}
    InputAirOk				AT %I* : BOOL;
		
	{attribute 'OPC.UA.DA.Access' := '1'}
	InputVacuumOk			AT %I* : BOOL;	
	
	{attribute 'OPC.UA.DA.Access' := '1'}
    InputSafetyDeviceOk		AT %I* : BOOL;
	
	{attribute 'OPC.UA.DA.Access' := '1'}
    InputLaserRelayOn		AT %I* : BOOL;
	
	{attribute 'OPC.UA.DA.Access' := '1'}
    InputMotionRelayOn		AT %I* : BOOL;
	
	{attribute 'OPC.UA.DA.Access' := '1'}
    InputWaferVacuumOk		AT %I* : BOOL;

	{attribute 'OPC.UA.DA.Access' := '1'}
    InputLiftPinUp			AT %I* : BOOL;
	
	{attribute 'OPC.UA.DA.Access' := '1'}
    InputLiftPinDown		AT %I* : BOOL;	
	
	{attribute 'OPC.UA.DA.Access' := '1'}
    InputPanel1Closed		AT %I* : BOOL;
	
	{attribute 'OPC.UA.DA.Access' := '1'}
    InputPanel2Closed		AT %I* : BOOL;
	
	{attribute 'OPC.UA.DA.Access' := '1'}
    InputPanel3Closed		AT %I* : BOOL;
	
	{attribute 'OPC.UA.DA.Access' := '1'}
    InputFrontCoverClosed	AT %I* : BOOL;
		
	{attribute 'OPC.UA.DA.Access' := '1'}
    InputWaferLoadSafetyDoorClosed	AT %I* : BOOL;
	
	{attribute 'OPC.UA.DA.Access' := '1'}
	InputDoorslitClosed				AT %I* : BOOL;
	
	{attribute 'OPC.UA.DA.Access' := '1'}
	InputDoorslitOpened				AT %I* : BOOL;
	
	
	(** Physical outputs **)	
	
	OutputLiftPinUp			AT %Q* : BOOL;	
	OutputLiftPinDown		AT %Q* : BOOL;
	OutputMotionEnable		AT %Q* : BOOL;
	OutputDoorslitMotorOn	AT %Q* : BOOL;
	OutputDoorslitMotorOpen	AT %Q* : BOOL;
	OutputVacuumOff			AT %Q* : BOOL;
	OutputCdaOff			AT %Q* : BOOL;
	OutputCounterBalanceOn	AT %Q* : BOOL;
	OutputHightThroughput	AT %Q* : BOOL;
	OutputMppcActivate		AT %Q* : BOOL := TRUE;	
	OutputCoolingFanFrontPanel AT %Q* : BOOL;
	OutputCoolingFanBackPanel  AT %Q* : BOOL;
END_STRUCT
END_TYPE

// ---- PMShared/Hardware/Devices/Chambers/Configs/Lightspeed/IoSafetyLS.TcDUT
{attribute 'OPC.UA.DA' := '1'}
TYPE IoSafetyLS :
STRUCT
	(** Physical inputs safety **)	
	
	{attribute 'OPC.UA.DA.Access' := '1'}
    InputSafetyIsShutterOk	AT %I* : BOOL;	

	{attribute 'OPC.UA.DA.Access' := '1'}
    InputSafetyIsExtPanelsInterlockOk	AT %I* : BOOL;
	
	{attribute 'OPC.UA.DA.Access' := '1'}
    InputSafetyIsOpticalBoxInterlockOk	AT %I* : BOOL;
	
	{attribute 'OPC.UA.DA.Access' := '1'}
    InputSafetyIsLaserContactorOk	AT %I* : BOOL;
	
	{attribute 'OPC.UA.DA.Access' := '1'}
    InputSafetyIsMotionContactorOk	AT %I* : BOOL;	
		
END_STRUCT
END_TYPE

// ---- PMShared/Hardware/Devices/Chambers/Configs/Lightspeed/LightspeedChamberConfig.TcDUT
TYPE LightspeedChamberConfig EXTENDS DeviceConfiguration :
STRUCT
	{attribute 'OPC.UA.DA' := '0'}
	Version : UINT;
	{attribute 'OPC.UA.DA' := '0'}
	Description: STRING;
END_STRUCT
END_TYPE

// ---- PMShared/Hardware/Devices/Chambers/Configs/PhotoLum/EFeedbackMsgPhotoLumChamber.TcDUT
{attribute 'qualified_only'}
{attribute 'strict'}
TYPE EFeedbackMsgPhotoLumChamber :
(
	InterlockPanelsMsg := 20,
	SlitDoorPositionMsg := 30,
	SlitDoorOpenPositionMsg,
	SlitDoorClosePositionMsg
);
END_TYPE

// ---- PMShared/Hardware/Devices/Chambers/Configs/PhotoLum/IoChamberPhotoLum.TcDUT
{attribute 'OPC.UA.DA' := '1'}
TYPE IoChamberPhotoLum :
STRUCT
	(** Physical inputs **)					
	InputOpenSlitDoor	AT %I* : BOOL;
    InputCloseSlitDoor	AT %I* : BOOL;
	
	(** Physical outputs **)	
	OutputOpenSlitDoor	AT %Q* : BOOL;	
	OutputCloseSlitDoor	AT %Q* : BOOL;

	OutputEnableCamera AT %Q* : BOOL;
	
	EfemInterlockSlitDoor AT %Q* : BOOL;
	EfemInterlockArmExtendedEnable AT %Q* : BOOL;
END_STRUCT
END_TYPE

// ---- PMShared/Hardware/Devices/Chambers/Configs/PhotoLum/PhotoLumChamberConfig.TcDUT
TYPE PhotoLumChamberConfig EXTENDS DeviceConfiguration :
STRUCT
	{attribute 'OPC.UA.DA' := '0'}
	Version : UINT;
	{attribute 'OPC.UA.DA' := '0'}
	Description: STRING;
	{attribute 'OPC.UA.DA' := '0'}
	Interlock : ARRAY [0..const.PHOTOLUM_NUMBER_INTERLOCK_PANELS - 1] OF Interlock;
END_STRUCT
END_TYPE

// ---- PMShared/Hardware/Devices/Chambers/Configs/PSD/EFeedbackMsgPsdChamber.TcDUT
{attribute 'qualified_only'}
{attribute 'strict'}
TYPE EFeedbackMsgPsdChamber :
(
	InterlockPanelsMsg := 20,	
	SlitDoorPositionMsg := 30,
	SlitDoorOpenPositionMsg,
	SlitDoorClosePositionMsg,		
	CdaValveIsOpenMsg,
	RefreshingMsg
);
END_TYPE

// ---- PMShared/Hardware/Devices/Chambers/Configs/PSD/IoChamberPsd.TcDUT
{attribute 'OPC.UA.DA' := '1'}
TYPE IoChamberPsd :
STRUCT		
	(** Physical inputs **)					
	InputOpenSlitDoor	AT %I* : BOOL;
    InputCloseSlitDoor	AT %I* : BOOL;
	
	(** Physical outputs **)	
	OutputOpenSlitDoor	AT %Q* : BOOL;	
	OutputCloseSlitDoor	AT %Q* : BOOL;

	OutputEnableCameraFS AT %Q* : BOOL;
	OutputEnableCameraBS AT %Q* : BOOL;		
	OutputCdaPneumaticValve AT %Q* :BOOL;		
END_STRUCT
END_TYPE

// ---- PMShared/Hardware/Devices/Chambers/Configs/PSD/PsdChamberConfig.TcDUT
TYPE PsdChamberConfig EXTENDS DeviceConfiguration :
STRUCT
	{attribute 'OPC.UA.DA' := '0'}
	Version : UINT;
	{attribute 'OPC.UA.DA' := '0'}
	Description: STRING;
	{attribute 'OPC.UA.DA' := '0'}
	Interlock : ARRAY [0..Const.PSD_NUMBER_INTERLOCK_PANELS] OF Interlock;
END_STRUCT
END_TYPE

// ---- PMShared/Hardware/Devices/Chambers/Configs/PSD/SensorId.TcDUT
{attribute 'qualified_only'}
{attribute 'strict'}
TYPE SensorID :
(
	None := 1,
	Frontside := 2,
	Backside := 4
);
END_TYPE

// ---- PMShared/Hardware/Devices/Chucks/Configs/ChuckConfigs.TcDUT
TYPE ChuckConfigs :
STRUCT
	PsdChuckConfig : PsdChuckConfig;
	PhotoLumChuckConfig : PhotoLumChuckConfig;
END_STRUCT
END_TYPE

// ---- PMShared/Hardware/Devices/Chucks/Configs/EFeedbackMsgChuckBase.TcDUT
{attribute 'qualified_only'}
{attribute 'strict'}
TYPE EFeedbackMsgChuckBase :
(
	IsInLoadingPositionMsg := 10
);
END_TYPE

// ---- PMShared/Hardware/Devices/Chucks/Configs/EMaterialPresence.TcDUT
{attribute 'qualified_only'}
{attribute 'strict'}
TYPE EMaterialPresence :
(
	Unknown := 0,
	Present,
	NotPresent
);
END_TYPE

// ---- PMShared/Hardware/Devices/Chucks/Configs/EWaferSize.TcDUT
{attribute 'qualified_only'}
{attribute 'strict'}
{attribute 'to_string'}
TYPE EWaferSize :
(
	Unknown := 0,
	_50mm := 50,
	_100mm := 100,
	_150mm := 150,
	_200mm := 200,
	_300mm := 300
);
END_TYPE

// ---- PMShared/Hardware/Devices/Chucks/Configs/PhotLum/EFeedbackMsgPhotoLumChuck.TcDUT
{attribute 'qualified_only'}
{attribute 'strict'}
TYPE EFeedbackMsgPhotoLumChuck :
(
	WaferPresenceMsg := 10,
	IsInLoadingPositionMsg
);
END_TYPE

// ---- PMShared/Hardware/Devices/Chucks/Configs/PhotLum/IoChuckPhotoLum.TcDUT
TYPE IoChuckPhotoLum :
STRUCT		
	OutputVaccum100mm  AT %Q* : BOOL;
	OutputVaccum150mm AT %Q* : BOOL;		
	OutputVaccum200mm AT %Q* :BOOL;		
END_STRUCT
END_TYPE

// ---- PMShared/Hardware/Devices/Chucks/Configs/PhotLum/PhotoLumChuckConfig.TcDUT
TYPE PhotoLumChuckConfig EXTENDS DeviceConfiguration :
STRUCT
	{attribute 'OPC.UA.DA' := '0'}
	Version : UINT;
	{attribute 'OPC.UA.DA' := '0'}
	Description: STRING;			
	{attribute 'OPC.UA.DA' := '0'}
	WaferPresenceSensor : ARRAY [0..Const.PHOTOLUM_NUMBER_WAFER_PRESENCE_SENSORS - 1] OF WaferPresenceSensor;
END_STRUCT
END_TYPE

// ---- PMShared/Hardware/Devices/Chucks/Configs/PSD/EFeedbackMsgPsdChuck.TcDUT
{attribute 'qualified_only'}
{attribute 'strict'}
TYPE EFeedbackMsgPsdChuck :
(
	WaferPresenceMsg := 10
);
END_TYPE

// ---- PMShared/Hardware/Devices/Chucks/Configs/PSD/IoChuckPsd.TcDUT
TYPE IoChuckPsd :
STRUCT				
END_STRUCT
END_TYPE

// ---- PMShared/Hardware/Devices/Chucks/Configs/PSD/PsdChuckConfig.TcDUT
TYPE PsdChuckConfig EXTENDS DeviceConfiguration :
STRUCT
	{attribute 'OPC.UA.DA' := '0'}
	Version : UINT;
	{attribute 'OPC.UA.DA' := '0'}
	Description: STRING;			
	{attribute 'OPC.UA.DA' := '0'}
	WaferPresenceSensor : ARRAY [0..Const.PSD_NUMBER_WAFER_PRESENCE_SENSORS - 1] OF WaferPresenceSensor;
END_STRUCT
END_TYPE

// ---- PMShared/Hardware/Devices/DistanceSensors/Configs/DistanceSensorConfigs.TcDUT
TYPE DistanceSensorConfigs :
STRUCT
	MicroEpsilonDistanceSensorConfig : MicroEpsilonDistanceSensorConfig;
END_STRUCT
END_TYPE

// ---- PMShared/Hardware/Devices/DistanceSensors/Configs/MicroEpsilon/EFeedbackMsgMicroEpsilonDistanceSensor.TcDUT
{attribute 'qualified_only'}
{attribute 'strict'}
TYPE EFeedbackMsgMicroEpsilonDistanceSensor :
(
	StateMsg := 1,
	StatusMsg := 2,
	IsAliveMsg := 3,
	DistanceMsg := 10,
	IdMsg,
	CustomMsg
);
END_TYPE

// ---- PMShared/Hardware/Devices/DistanceSensors/Configs/MicroEpsilon/MicroEpsilonDistanceSensorConfig.TcDUT
TYPE MicroEpsilonDistanceSensorConfig EXTENDS DeviceConfiguration :
STRUCT
END_STRUCT
END_TYPE

// ---- PMShared/Hardware/Devices/DistanceSensors/Configs/MicroEpsilon/IoMicroEpsilonDistanceSensor.TcDUT
TYPE IoMicroEpsilonDistanceSensor :
STRUCT
	InputMicroEpsilonDistanceSensor AT %I* : REAL;	
END_STRUCT
END_TYPE

// ---- PMShared/Hardware/Devices/FastAttenuation/Configs/FastAttenuationConfigs.TcDUT
TYPE FastAttenuationConfigs :
STRUCT
	Std900FastAttenuationConfig : Std900FastAttenuationConfig;
END_STRUCT
END_TYPE

// ---- PMShared/Hardware/Devices/FastAttenuation/Configs/Parallax/EFeedbackMsgStd900.TcDUT
{attribute 'qualified_only'}
{attribute 'strict'}
TYPE EFeedbackMsgStd900 :
(
	PositionMsg := 10
);
END_TYPE

// ---- PMShared/Hardware/Devices/FastAttenuation/Configs/Parallax/IoStd900.TcDUT
TYPE IoStd900 :
STRUCT	
	OutputPwm		AT %Q* : UINT;
	OutputPeriodPwm	AT %Q* : UINT;	
END_STRUCT
END_TYPE

// ---- PMShared/Hardware/Devices/FastAttenuation/Configs/Parallax/Std900FastAttenuationConfig.TcDUT
TYPE Std900FastAttenuationConfig EXTENDS DeviceConfiguration :
STRUCT
END_STRUCT
END_TYPE

// ---- PMShared/Hardware/Devices/Ffus/Astrofan/Loop/FfuSpeedMatrix/Ffumatrixconfig.TcDUT
TYPE Ffumatrixconfig :
STRUCT
	Enable : BOOL;
	FfuMatrix : ARRAY [0 .. Constants.speedMatrixSize] OF FfuSpeed;
END_STRUCT
END_TYPE

// ---- PMShared/Hardware/Devices/Ffus/Astrofan/Loop/FfuSpeedMatrix/FfuSpeed.TcDUT
TYPE FfuSpeed :
STRUCT
	NonScaledSpeedValue	: UINT;
	ScaledSpeedValue	: UINT;
END_STRUCT
END_TYPE

// ---- PMShared/Hardware/Devices/Ffus/Configs/Astrofan/Astrofan612FfuConfig.TcDUT
TYPE Astrofan612FfuConfig EXTENDS DeviceConfiguration :
STRUCT
	SpeedMatrix	: FfuMatrixconfig;
	Loop : Astrofan612FfuLoopConfig;
END_STRUCT
END_TYPE

// ---- PMShared/Hardware/Devices/Ffus/Configs/Astrofan/Astrofan612FfuLoopConfig.TcDUT
TYPE Astrofan612FfuLoopConfig :
STRUCT
	IsEnabled : BOOL;
	FfuLoopStandardSetSpeed : UINT;
	FfuLoopPressureTimerSeconds : UINT;
	FfuLoopWarning 	: Astrofan612FfuEvent;
	FfuLoopAlarm 	: Astrofan612FfuEvent;
	FfuPressureMinimumValuePa : UINT;
	FfuPressureMaximumValuePa : UINT;
	FfuLoopSetSpeedHigherLimitPercent : UINT;
	FfuLoopSetSpeedLowerLimitPercent : UINT;
END_STRUCT
END_TYPE

// ---- PMShared/Hardware/Devices/Ffus/Configs/Astrofan/Astrofan612FfuEvent.TcDUT
TYPE Astrofan612FfuEvent :
STRUCT
	ThresholdPercent : UINT;
	TimerSeconds : UINT;
END_STRUCT
END_TYPE

// ---- PMShared/Hardware/Devices/Ffus/Configs/Astrofan/EFeedbackMsgAstrofan612.TcDUT
{attribute 'qualified_only'}
{attribute 'strict'}
TYPE EFeedbackMsgAstrofan612 :
(		
	StateMsg := 1,
	StatusMsg := 2,
	IsAliveMsg := 3,
	CurrentSpeedMsg := 10,
	TemperatureMsg,
	WarningRaisedMsg := 20,
	AlarmRaisedMsg,
	CustomMsg := 50
);
END_TYPE

// ---- PMShared/Hardware/Devices/Ffus/Configs/FfuConfigs.TcDUT
TYPE FfuConfigs :
STRUCT
	Astrofan612FfuConfig : Astrofan612FfuConfig;
END_STRUCT
END_TYPE

// ---- PMShared/Hardware/Devices/FiberSwitch/Configs/FiberSwitchConfigs.TcDUT
TYPE FiberSwitchConfigs :
STRUCT
	EOLFiberSwitchConfig : EOLFiberSwitchConfig;
END_STRUCT
END_TYPE

// ---- PMShared/Hardware/Devices/FiberSwitch/Configs/Leoni/EFeedbackMsgEol.TcDUT
{attribute 'qualified_only'}
{attribute 'strict'}
TYPE EFeedbackMsgEol :
(
	IdMsg := 10,
    CustomMsg
);
END_TYPE

// ---- PMShared/Hardware/Devices/FiberSwitch/Configs/Leoni/EOLFiberSwitchConfig.TcDUT
TYPE EOLFiberSwitchConfig EXTENDS DeviceConfiguration :
STRUCT
	SerialCommunication : SerialCommunication;
END_STRUCT
END_TYPE

// ---- PMShared/Hardware/Devices/Ionizers/Configs/IonizerAlarm.TcDUT
{attribute 'OPC.UA.DA' := '0'}
TYPE IonizerAlarm :
STRUCT
	Name : STRING;
	Description : STRING;
	AlarmID : UINT;
	Triggered AT %I* : BOOL;
END_STRUCT
END_TYPE

// ---- PMShared/Hardware/Devices/Ionizers/Configs/IonizerConfigs.TcDUT
TYPE IonizerConfigs :
STRUCT
	SJH108IonizerConfig : SJH108IonizerConfig;
END_STRUCT
END_TYPE

// ---- PMShared/Hardware/Devices/Ionizers/Configs/Keyence/EFeedbackMsgSJH108.TcDUT
{attribute 'qualified_only'}
{attribute 'strict'}
TYPE EFeedbackMsgSJH108 :
(
	StateMsg := 1,
	StatusMsg := 2,
	IsAliveMsg := 3,
	AlarmMsg := 10,
	AirValveIsOpenMsg,
	StaticEliminationInterruptMsg,
	RefreshingMsg
);
END_TYPE

// ---- PMShared/Hardware/Devices/Ionizers/Configs/Keyence/IoSJH108A.TcDUT
{attribute 'OPC.UA.DA' := '1'}
TYPE IoSJH108A :
STRUCT					
	OutputOpenAirValve	AT %Q* : BOOL;	
	OutputStaticEliminationInterrupt AT %Q* : BOOL;
END_STRUCT
END_TYPE

// ---- PMShared/Hardware/Devices/Ionizers/Configs/Keyence/SJH108IonizerConfig.TcDUT
TYPE SJH108IonizerConfig EXTENDS DeviceConfiguration :
STRUCT
	{attribute 'OPC.UA.DA' := '0'}
	IonizerAlarm : ARRAY [0..IonizerConst.NUMBER_ALARMS] OF IonizerAlarm;
END_STRUCT
END_TYPE

// ---- PMShared/Hardware/Devices/Lasers/Configs/Base/HoursStruct.TcDUT
TYPE HoursStruct :
STRUCT
END_STRUCT
END_TYPE

// ---- PMShared/Hardware/Devices/Lasers/Configs/Coherent/EFeedbackMsgSapphire488.TcDUT
{attribute 'qualified_only'}
{attribute 'strict'}
TYPE EFeedbackMsgSapphire488 :
(
	PowerMsg := 10,
    InterlockStatusMsg,
    BasePlateTemperatureMsg,
    ControllerTemperatureMsg,
	DiodeSetTemperatureMsg,
	MeasuredTemperatureMsg,
	LaserHeadReachedDiodeCurrentLimitMsg,
    IdMsg,
    CustomMsg
);
END_TYPE

// ---- PMShared/Hardware/Devices/Lasers/Configs/Coherent/Sapphire488LaserConfig.TcDUT
TYPE Sapphire488LaserConfig EXTENDS DeviceConfiguration :
STRUCT
	SerialCommunication : SerialCommunication;
END_STRUCT
END_TYPE

// ---- PMShared/Hardware/Devices/Lasers/Configs/LaserConfigs.TcDUT
TYPE LaserConfigs :
STRUCT
	SMD12LaserConfig : SMD12LaserConfig;
	Piano450LaserConfig : Piano450LaserConfig;
	Sapphire488LaserConfig : Sapphire488LaserConfig;
END_STRUCT
END_TYPE

// ---- PMShared/Hardware/Devices/Lasers/Configs/Leukos/EControlModePiano450.TcDUT
{attribute 'qualified_only'}
{attribute 'strict'}
TYPE EControlModePiano450 :
(
	PowerMode
);
END_TYPE

// ---- PMShared/Hardware/Devices/Lasers/Configs/Leukos/EFeedbackMsgPiano450.TcDUT
{attribute 'qualified_only'}
{attribute 'strict'}
TYPE EFeedbackMsgPiano450 :
(		
	StateMsg := 1,
	StatusMsg := 2,
	IsAliveMsg := 3,
	PowerMsg := 10,	
    InterlockStatusMsg,
    LaserTemperatureMsg,
    CrystalTemperatureMsg,
	RunningTimeLaserOnMsg,
    RunningTimeElectroOnMsg,
    CustomMsg	
);
END_TYPE

// ---- PMShared/Hardware/Devices/Lasers/Configs/Leukos/Piano450LaserConfig.TcDUT
TYPE Piano450LaserConfig EXTENDS DeviceConfiguration :
STRUCT
	SerialCommunication : SerialCommunication;
END_STRUCT
END_TYPE

// ---- PMShared/Hardware/Devices/Lasers/Configs/Quantum/EControlModeSmd12.TcDUT
{attribute 'qualified_only'}
{attribute 'strict'}
TYPE EControlModeSmd12 :
(
	CurrentMode, 
	PowerMode
);
END_TYPE

// ---- PMShared/Hardware/Devices/Lasers/Configs/Quantum/EFeedbackMsgSMD12.TcDUT
{attribute 'qualified_only'}
{attribute 'strict'}
TYPE EFeedbackMsgSMD12 :
(
	PowerMsg := 10,
    InterlockStatusMsg,
    LaserTemperatureMsg,
    PsuTemperatureMsg,
    IdMsg,
    CustomMsg
);
END_TYPE

// ---- PMShared/Hardware/Devices/Lasers/Configs/Quantum/SMD12LaserConfig.TcDUT
TYPE SMD12LaserConfig EXTENDS DeviceConfiguration :
STRUCT
	SerialCommunication : SerialCommunication;
END_STRUCT
END_TYPE

// ---- PMShared/Hardware/Devices/Lights/Configs/Evosens/EvosensLightConfig.TcDUT
TYPE EvosensLightConfig EXTENDS DeviceConfiguration :
STRUCT
	SerialCommunication : SerialCommunication;
END_STRUCT
END_TYPE

// ---- PMShared/Hardware/Devices/Lights/Configs/Evosens/EFeedbackMsgEvosensLight.TcDUT
{attribute 'qualified_only'}
{attribute 'strict'}
TYPE EFeedbackMsgEvosensLight :
(		
	StateMsg := 1,
	StatusMsg := 2,
	IsAliveMsg := 3,
	SwitchOnMsg := 10,
    PowerMsg,
    IntensityMsg,
    TemperatureMsg,
    LightSourcesMsg,
    TimeLightSourceMsg,
    CustomMsg := 50
);
END_TYPE

// ---- PMShared/Hardware/Devices/Lights/Configs/Arduino/EFeedbackMsgArduinoLight.TcDUT
{attribute 'qualified_only'}
{attribute 'strict'}
TYPE EFeedbackMsgArduinoLight :
(		
	StateMsg := 1,
	StatusMsg := 2,
	IsAliveMsg := 3,
	SwitchOnMsg := 10,
    PowerMsg,
    IntensityMsg,
    TemperatureMsg,
    LightSourcesMsg,
    TimeLightSourceMsg,
    CustomMsg := 50
);
END_TYPE

// ---- PMShared/Hardware/Devices/Lights/Configs/Arduino/ArduinoLightConfig.TcDUT
TYPE ArduinoLightConfig EXTENDS DeviceConfiguration :
STRUCT
	SerialCommunication : SerialCommunication;
END_STRUCT
END_TYPE

// ---- PMShared/Hardware/Devices/Lights/Configs/LightConfigs.TcDUT
TYPE LightConfigs :
STRUCT	
	ArduinoLightConfig : ArduinoLightConfig;
	EvosensLightConfig : EvosensLightConfig;
END_STRUCT
END_TYPE

// ---- PMShared/Hardware/Devices/MPPCs/Configs/Hamamatsu/C13336MppcConfig.TcDUT
TYPE C13336MppcConfig EXTENDS DeviceConfiguration :
STRUCT
	SerialCommunication : SerialCommunication;
END_STRUCT
END_TYPE

// ---- PMShared/Hardware/Devices/MPPCs/Configs/Hamamatsu/EFeedbackMsgC13336.TcDUT
{attribute 'qualified_only'}
{attribute 'strict'}
TYPE  EFeedbackMsgC13336 :
(	
	MonitorInfoStatusMsg := 10,
	OutputCurrentMsg,
	OutputVoltageMsg,
	OutputVoltageSettingMsg,
	StatusMsg,
	TemperatureMsg,
	SensorTemperatureMsg,
	PowerFctReadMSg,
	TempCorrectionFactorReadMsg,
	FirmwareMsg,
    IdentifierMsg,
    CustomMsg,
	StateSignalsMsg	
);
END_TYPE

// ---- PMShared/Hardware/Devices/MPPCs/Configs/Hamamatsu/EMppcCollector.TcDUT
{attribute 'qualified_only'}
{attribute 'strict'}
{attribute 'to_string'}
TYPE EMppcCollector :
(
	Unknown := 0,
    WIDE,
    NARROW
);
END_TYPE

// ---- PMShared/Hardware/Devices/MPPCs/Configs/Hamamatsu/EMppcStateModule.TcDUT
{attribute 'qualified_only'}
{attribute 'strict'}
{attribute 'to_string'}
TYPE EMppcStateModule :
(
	UNRECOVERABLE_ERROR := 0,
	AWAITING_COOLING_TEMP_STABLE,
	AWAITING_HIGH_VOLTAGE_POWER_SUPPLY_STABLE,
	MODULE_OPERATING_NORMAL 
);
END_TYPE

// ---- PMShared/Hardware/Devices/MPPCs/Configs/Hamamatsu/IoC13336Mppc.TcDUT
TYPE IoC13336Mppc :
STRUCT	
	(** One relay manage 2 MPPCs -> The wide MPPC output is physically and only connected. It also manages the relay of the Narrow MPPC output **)
	OutputMppcRelayPower : BOOL; 
END_STRUCT
END_TYPE

// ---- PMShared/Hardware/Devices/MPPCs/Configs/MppcConfigs.TcDUT
TYPE MppcConfigs :
STRUCT
	C13336MppcConfigWide   : C13336MppcConfig;
	C13336MppcConfigNarrow : C13336MppcConfig;
END_STRUCT
END_TYPE

// ---- PMShared/Hardware/Devices/OpticalPowermeters/Configs/OpticalPowermeterConfigs.TcDUT
TYPE OpticalPowermeterConfigs :
STRUCT
	PM101OpticalPowermeterConfigHs : PM101OpticalPowermeterConfig;
	PM101OpticalPowermeterConfigHt : PM101OpticalPowermeterConfig;
END_STRUCT
END_TYPE

// ---- PMShared/Hardware/Devices/OpticalPowermeters/Configs/Thorlabs/EFeedbackMsgPM101.TcDUT
{attribute 'qualified_only'}
{attribute 'strict'}
TYPE EFeedbackMsgPM101 :
(
	PowerMsg := 10,
	CurrentMsg,
	IdentifierMsg,
	ResponsivityMsg,
	DarkOffsetMsg,
	DarkAdjustStateMsg,
	CustomMsg,	 
	SensorTypeMsg,	
	WavelengthMsg,		     
    BeamDiameterMsg,
	SensorAttenuationMsg,
    WavelengthRangeMsg,
    MaxPowerMsg,
    MinPowerMsg,
	CalibMsg
);
END_TYPE

// ---- PMShared/Hardware/Devices/OpticalPowermeters/Configs/Thorlabs/EPowerIlluminationFlow.TcDUT
{attribute 'qualified_only'}
{attribute 'strict'}
{attribute 'to_string'}
TYPE EPowerIlluminationFlow :
(
	HS := 1,
	HT
);
END_TYPE

// ---- PMShared/Hardware/Devices/OpticalPowermeters/Configs/Thorlabs/IoControlPM101.TcDUT
TYPE IoControlPM101 :
STRUCT
	{attribute 'OPC.UA.DA.Access' := '1'}
    InputGeneral_1		AT %I* : BOOL;
	
	{attribute 'OPC.UA.DA.Access' := '1'}
    InputGeneral_2		AT %I* : BOOL;
	
	
	(** Physical outputs **)
	OutputMeasurementRange	AT %Q* : LREAL;
END_STRUCT
END_TYPE

// ---- PMShared/Hardware/Devices/OpticalPowermeters/Configs/Thorlabs/PM101OpticalPowermeterConfig.TcDUT
TYPE PM101OpticalPowermeterConfig EXTENDS DeviceConfiguration :
STRUCT
	SerialCommunication : SerialCommunication;
	Sensor : PowermeterSensor;
END_STRUCT
END_TYPE

// ---- PMShared/Hardware/Devices/OpticalPowermeters/Thorlabs/PM101/Messages/BeamDiameterMsg.TcDUT
{attribute 'OPC.UA.DA' := '1'}
{attribute 'OPC.UA.DA.StructuredType' := '1'}
TYPE BeamDiameterMsg :
STRUCT
	Id : EPowerIlluminationFlow;
	BeamDiameter : INT;
END_STRUCT
END_TYPE

// ---- PMShared/Hardware/Devices/OpticalPowermeters/Thorlabs/PM101/Messages/AttenuationMsg.TcDUT
{attribute 'OPC.UA.DA' := '1'}
{attribute 'OPC.UA.DA.StructuredType' := '1'}
TYPE AttenuationMsg :
STRUCT
	Id : EPowerIlluminationFlow;
	Attenuation : UINT;
END_STRUCT
END_TYPE

// ---- PMShared/Hardware/Devices/OpticalPowermeters/Thorlabs/PM101/Messages/SensorTypeMsg.TcDUT
{attribute 'OPC.UA.DA' := '1'}
{attribute 'OPC.UA.DA.StructuredType' := '1'}
TYPE SensorTypeMsg :
STRUCT
	Id : EPowerIlluminationFlow;
	SensorType : STRING(255);
END_STRUCT
END_TYPE

// ---- PMShared/Hardware/Devices/OpticalPowermeters/Thorlabs/PM101/Messages/ResponsivityMsg.TcDUT
{attribute 'OPC.UA.DA' := '1'}
{attribute 'OPC.UA.DA.StructuredType' := '1'}
TYPE ResponsivityMsg :
STRUCT
	Id : EPowerIlluminationFlow;
	Responsivity : LREAL;
END_STRUCT
END_TYPE

// ---- PMShared/Hardware/Devices/OpticalPowermeters/Thorlabs/PM101/Messages/CustomMsg.TcDUT
{attribute 'OPC.UA.DA' := '1'}
{attribute 'OPC.UA.DA.StructuredType' := '1'}
TYPE CustomMsg :
STRUCT	
	Id : EPowerIlluminationFlow;
	Custom : STRING(255);
END_STRUCT
END_TYPE

// ---- PMShared/Hardware/Devices/OpticalPowermeters/Thorlabs/PM101/Messages/IdentifierMsg.TcDUT
{attribute 'OPC.UA.DA' := '1'}
{attribute 'OPC.UA.DA.StructuredType' := '1'}
TYPE IdentifierMsg :
STRUCT
	Id : EPowerIlluminationFlow;
	Identifier : STRING(255);
END_STRUCT
END_TYPE

// ---- PMShared/Hardware/Devices/OpticalPowermeters/Thorlabs/PM101/Messages/MaxPowerMsg.TcDUT
{attribute 'OPC.UA.DA' := '1'}
{attribute 'OPC.UA.DA.StructuredType' := '1'}
TYPE MaxPowerMsg :
STRUCT
	Id : EPowerIlluminationFlow;
	MaxPower : LREAL;
END_STRUCT
END_TYPE

// ---- PMShared/Hardware/Devices/OpticalPowermeters/Thorlabs/PM101/Messages/MinPowerMsg.TcDUT
{attribute 'OPC.UA.DA' := '1'}
{attribute 'OPC.UA.DA.StructuredType' := '1'}
TYPE MinPowerMsg :
STRUCT
	Id : EPowerIlluminationFlow;
	MinPower : LREAL;
END_STRUCT
END_TYPE

// ---- PMShared/Hardware/Devices/OpticalPowermeters/Thorlabs/PM101/Messages/PowerMsg.TcDUT
TYPE PowerMsg :
STRUCT
	Id : EPowerIlluminationFlow;
	Power : LREAL;
	PowerCal_mW : LREAL; 
END_STRUCT
END_TYPE

// ---- PMShared/Hardware/Devices/OpticalPowermeters/Thorlabs/PM101/Messages/WavelengthMsg.TcDUT
{attribute 'OPC.UA.DA' := '1'}
{attribute 'OPC.UA.DA.StructuredType' := '1'}
TYPE WavelengthMsg :
STRUCT
	Id : EPowerIlluminationFlow;
	Wavelength : INT;
END_STRUCT
END_TYPE

// ---- PMShared/Hardware/Devices/OpticalPowermeters/Thorlabs/PM101/Messages/WavelengthRangeMsg.TcDUT
{attribute 'OPC.UA.DA' := '1'}
{attribute 'OPC.UA.DA.StructuredType' := '1'}
TYPE WavelengthRangeMsg :
STRUCT
	Id : EPowerIlluminationFlow;
	WavelengthRange : STRING(255);
END_STRUCT
END_TYPE

// ---- PMShared/Hardware/Devices/PolarisationFilters/Configs/PolarisationFilterConfigs.TcDUT
TYPE PolarisationFilterConfigs :
STRUCT
	FW212CPolarisationFilterConfig : FW212CPolarisationFilterConfig;
	ELL14KPolarisationFilterConfig : ELL14KPolarisationFilterConfig;
END_STRUCT
END_TYPE

// ---- PMShared/Hardware/Devices/PolarisationFilters/Configs/Thorlabs/ELL14K/EFeedbackMsgPolarisationELL14K.TcDUT
{attribute 'qualified_only'}
{attribute 'strict'}
TYPE EFeedbackMsgPolarisationELL14K :
(
	PositionMsg := 10,
    IdMsg,
	CalibMsg,
    CustomMsg
);
END_TYPE

// ---- PMShared/Hardware/Devices/PolarisationFilters/Configs/Thorlabs/ELL14K/ELL14KPolarisationFilterConfig.TcDUT
TYPE ELL14KPolarisationFilterConfig EXTENDS DeviceConfiguration :
STRUCT
	SerialCommunication : SerialCommunication;
END_STRUCT
END_TYPE

// ---- PMShared/Hardware/Devices/PolarisationFilters/Configs/Thorlabs/EPolar.TcDUT
{attribute 'qualified_only'}
{attribute 'strict'}
{attribute 'to_string'}
TYPE EPolar :
(
	Unknown := 0,
	S_Polar,
	P_Polar
);
END_TYPE

// ---- PMShared/Hardware/Devices/PolarisationFilters/Configs/Thorlabs/FW212C/EFeedbackMsgPolarisationFW212C.TcDUT
{attribute 'qualified_only'}
{attribute 'strict'}
TYPE EFeedbackMsgPolarisationFW212C :
(
	CheckConnectionMsg := 10,
    PositionMsg,
    PositionCountMsg,
    IdMsg,
    CustomMsg
);
END_TYPE

// ---- PMShared/Hardware/Devices/PolarisationFilters/Configs/Thorlabs/FW212C/FW212CPolarisationFilterConfig.TcDUT
TYPE FW212CPolarisationFilterConfig EXTENDS DeviceConfiguration :
STRUCT
	SerialCommunication : SerialCommunication;
END_STRUCT
END_TYPE

// ---- PMShared/Hardware/Devices/Chambers/Configs/ChamberConfigs.TcDUT
TYPE ChamberConfigs :
STRUCT
	PsdChamberConfig : PsdChamberConfig;
	LightspeedChamberConfig : LightspeedChamberConfig;	
	PhotoLumChamberConfig : PhotoLumChamberConfig;
END_STRUCT
END_TYPE

// ---- PMShared/Hardware/Devices/Rfids/Configs/Balluff/BisL405RfidConfig.TcDUT
TYPE BisL405RfidConfig EXTENDS DeviceConfiguration :
STRUCT
	{attribute 'OPC.UA.DA' := '0'}
	Version : UINT;
	{attribute 'OPC.UA.DA' := '0'}
	Description: STRING;
END_STRUCT
END_TYPE

// ---- PMShared/Hardware/Devices/Rfids/Configs/Balluff/EFeedbackMsgBisL405.TcDUT
{attribute 'qualified_only'}
{attribute 'strict'}
TYPE EFeedbackMsgBisL405 :
(
	DataCarrierMsg := 10
);
END_TYPE

// ---- PMShared/Hardware/Devices/Rfids/Configs/Balluff/IoBisL405Rfid.TcDUT
{attribute 'OPC.UA.DA.Access' := '0'}
TYPE IoBisL405Rfid :
STRUCT
    TagPresent AT %I* : BOOL;
    Strobe AT %I* : BOOL;
	DataOutput0 AT %I* : BOOL;
	DataOutput1 AT %I* : BOOL;
	DataOutput2 AT %I* : BOOL;
	DataOutput3 AT %I* : BOOL;
	DataOutput4 AT %I* : BOOL;
	DataOutput5 AT %I* : BOOL;
	DataOutput6 AT %I* : BOOL;
	DataOutput7 AT %I* : BOOL;
	
	Address AT %Q* : BOOL;
	Restart AT %Q* : BOOL;
END_STRUCT
END_TYPE

// ---- PMShared/Hardware/Devices/Rfids/Configs/RfidConfigs.TcDUT
TYPE RfidConfigs :
STRUCT
	BisL405RfidConfig : BisL405RfidConfig;
END_STRUCT
END_TYPE

// ---- PMShared/Hardware/Devices/Safety/Configs/Interlock.TcDUT
{attribute 'OPC.UA.DA' := '0'}
TYPE Interlock :
STRUCT
	Name : STRING;
	Description : STRING;
	InterlockID : UINT;
	State AT %I* : BOOL;
END_STRUCT
END_TYPE

// ---- PMShared/Hardware/Devices/Screens/Configs/Densitron/DM430GNScreenConfig.TcDUT
TYPE DM430GNScreenConfig EXTENDS DeviceConfiguration :
STRUCT
	SerialCommunication : SerialCommunication;
END_STRUCT
END_TYPE

// ---- PMShared/Hardware/Devices/Screens/Configs/Densitron/EDisplayControlStep.TcDUT
{attribute 'qualified_only'}
{attribute 'strict'}
TYPE EDisplayControlStep :
(
	Percent_0 := 0,
	Percent_25 := 1,
	Percent_50 := 2,
	Percent_75 := 3,
	Percent_100 := 4
);
END_TYPE

// ---- PMShared/Hardware/Devices/Screens/Configs/Densitron/EFeedbackMsgDM430GN.TcDUT
{attribute 'qualified_only'}
{attribute 'strict'}
TYPE EFeedbackMsgDM430GN :
(
	StateMsg := 1,
	StatusMsg := 2,
	IsAliveMsg := 3,
	PowerStateMsg := 10,
	BacklightMsg,
	BrightnessMsg,
	ContrastMsg,
	FanAutoMsg,
	FanStepMsg,
	FanRpmMsg,
	TemperatureMsg,
	CustomMsg := 50
);
END_TYPE

// ---- PMShared/Hardware/Devices/Screens/Configs/Densitron/EScreenSide.TcDUT
{attribute 'qualified_only'}
{attribute 'strict'}
{attribute 'to_string'}
TYPE EScreenSide :
(
	Unknown := 0,
    Back,
    Front
);
END_TYPE

// ---- PMShared/Hardware/Devices/Screens/Configs/ScreenConfigs.TcDUT
TYPE ScreenConfigs :
STRUCT
	DM430GNScreenConfigFS : DM430GNScreenConfig;
	DM430GNScreenConfigBS : DM430GNScreenConfig;
END_STRUCT
END_TYPE

// ---- PMShared/Hardware/Devices/Shutters/Configs/Eopc/Sh10pilShutterConfig.TcDUT
TYPE Sh10pilShutterConfig EXTENDS DeviceConfiguration :
STRUCT	
END_STRUCT
END_TYPE

// ---- PMShared/Hardware/Devices/Shutters/Configs/Eopc/EFeedbackMsgSh10pil.TcDUT
{attribute 'qualified_only'}
{attribute 'strict'}
TYPE EFeedbackMsgSh10pil :
(
	ShutterIrisPositionMsg := 10
);
END_TYPE

// ---- PMShared/Hardware/Devices/Shutters/Configs/Eopc/IoSh10pilShutter.TcDUT
TYPE IoSh10pilShutter :
STRUCT
	InputMagneticSwitch1	AT %I* : BOOL;	
	InputMagneticSwitch2	AT %I* : BOOL;		
	OutputSwitchContactClosure	AT %Q* : BOOL;	
END_STRUCT
END_TYPE

// ---- PMShared/Hardware/Devices/Shutters/Configs/ShutterConfigs.TcDUT
TYPE ShutterConfigs :
STRUCT
	Ed12dssShutterConfig : Ed12dssShutterConfig;
	Sh10pilShutterConfig : Sh10pilShutterConfig;
END_STRUCT
END_TYPE

// ---- PMShared/Hardware/Devices/Shutters/Configs/Uniblitz/Ed12dssShutterConfig.TcDUT
TYPE Ed12dssShutterConfig EXTENDS DeviceConfiguration :
STRUCT	
END_STRUCT
END_TYPE

// ---- PMShared/Hardware/Devices/Shutters/Configs/Uniblitz/EFeedbackMsgEd12dss.TcDUT
{attribute 'qualified_only'}
{attribute 'strict'}
TYPE EFeedbackMsgEd12dss :
(
	ShutterIrisPositionMsg := 10
);
END_TYPE

// ---- PMShared/Hardware/Devices/Shutters/Configs/Uniblitz/IoEd12dssShutter.TcDUT
TYPE IoEd12dssShutter :
STRUCT	
	OutputSwitchContactClosure	AT %Q* : BOOL;	
	
	inputShutter1 AT %I* : BOOL;
	inputShutter2 AT %I* : BOOL;
END_STRUCT
END_TYPE

// ---- PMShared/Hardware/Interface/TrackExecution/TExecutionState.TcDUT
{attribute 'qualified_only'}
{attribute 'strict'}
{attribute 'to_string'}
TYPE TExecutionState :
(	
	Unknown := 0,
	Ready,
    Starting,
    Busy,
	Error,
	Warning
);
END_TYPE

// ---- Service/PMs/EFeedbackMsgPlc.TcDUT
{attribute 'qualified_only'}
{attribute 'strict'}
TYPE EFeedbackMsgPlc :
(
	SmokeDetectedMsg := 0,
	SmokeDetectorFaultMsg,
	VacuumDetectorMsg,
	AmsNetIdMsg
);
END_TYPE

// ---- Service/PMs/Lightspeed/Calibrate/LsCalibrateConfig.TcDUT
{attribute 'OPC.UA.DA' := '0'}
TYPE LsCalibrateConfig :
STRUCT
	HSPowermeter : HSPowermeter;
	HTPowermeter : HTPowermeter;
END_STRUCT
END_TYPE

// ---- Service/PMs/Lightspeed/Calibrate/PolarisationConfig.TcDUT
{attribute 'OPC.UA.DA' := '0'}
TYPE PolarisationConfig :
STRUCT
	PolarAngle_S : LREAL;
	PolarAngle_P : LREAL;
END_STRUCT
END_TYPE

// ---- Service/PMs/Lightspeed/Calibrate/ResponsivityConfig.TcDUT
{attribute 'OPC.UA.DA' := '0'}
TYPE ResponsivityConfig :
STRUCT
	Responsivity_mA_W : LREAL;
END_STRUCT
END_TYPE

// ---- Service/PMs/Lightspeed/Calibrate/RFactorBase.TcDUT
{attribute 'OPC.UA.DA' := '0'}
TYPE RFactorBase :
STRUCT
	RFactor_S : LREAL;
	RFactor_P : LREAL;
END_STRUCT
END_TYPE

// ---- Service/PMs/Lightspeed/Calibrate/RFactorSettings.TcDUT
{attribute 'OPC.UA.DA' := '0'}
TYPE RFactorSettings EXTENDS RFactorBase :
STRUCT
END_STRUCT
END_TYPE

// ---- Shared/Log/LogEventLevel.TcDUT
{attribute 'qualified_only'}
{attribute 'strict'}
TYPE LogEventLevel :
(	
    Verbose := 0,
    Debug,
    Information,
    Warning,
    Error,
    Fatal
);
END_TYPE

// ---- PMShared/Hardware/Devices/Axes/AxesConst.TcGVL
{attribute 'qualified_only'}
VAR_GLOBAL CONSTANT PERSISTENT
	AXIS_FILTER_WHEEL : STRING := '1';
	
	// FILTER WHEEL
	FW_DRIVING_CURRENT_IN_PERCENT : UINT := 90;
	FW_HOLDING_CURRENT_IN_PERCENT : UINT := 50;
	FW_LIMIT_SWITCH_MASK : UINT := 0;
END_VAR

// ---- PMShared/Hardware/Devices/Ffus/Astrofan/Constants.TcGVL
{attribute 'qualified_only'}
VAR_GLOBAL CONSTANT 
	speedMatrixSize : UINT := 10;
	 
END_VAR

// ---- PMShared/Hardware/Devices/Ionizers/Configs/IonizerConst.TcGVL
{attribute 'qualified_only'}
VAR_GLOBAL CONSTANT PERSISTENT
	NUMBER_ALARMS : UINT := 1;
END_VAR

// ---- Shared/GlobalVariables/Const.TcGVL
{attribute 'qualified_only'}
VAR_GLOBAL CONSTANT PERSISTENT
	APP_CONFIG_FILE_PATH : T_MaxString := 'C:\Unity\app.config';	
	APP_CONFIG_XPATH 	 : T_MaxString := '/AppConfig';
	
	SERIAL_COM_CHANNEL_1 : STRING := 'Com1';
	SERIAL_COM_CHANNEL_2 : STRING := 'Com2';
	
	ATTENUATION_AXIS : STRING := 'AttenuationAxis';
	POLARISATION_AXIS : STRING := 'PolarisationAxis';
	
	START_OF_TEXT : STRING := '$02';			
	CARRIAGE_RETURN : STRING := '$0D';
	LINE_FEED : STRING := '$0A';
	CR_LF : STRING := '$0D$0A';
	LF_CR : STRING := '$0A$0D';
	ETX_CHKSUM_CR : STRING := '$03$45$43$0D';
		
	PULSES_PER_DEG : REAL := 143360.0 / 360.0;	
	
	ELL9_TRAVEL : UINT := 93; 
	ELL9_NUMBER_POS : UINT := 4;
	
	ELL6_TRAVEL : UINT := 31; 
	ELL6_NUMBER_POS : UINT := 2;
	
	ACTIVE_TIME_COOLING_FAN : TIME := T#1M;
	
	STD900_INTERVAL : UINT := 20000; // the servo needs to receive a pulse every 20000 µs.
	STD900_LOW_LIMIT : UINT := 1175; // µs (is equivalent to 750 µs)
	STD900_HIGHT_LIMIT : UINT := 3200; // µs (is equivalent to 2250 µs)
	STD900_MIN_ANGLE : UINT := 0;
	STD900_MAX_ANGLE : UINT := 180;
	
	POWERMETER_SENSOR_NAME_S150C : STRING := 'S150C';
	POWERMETER_SENSOR_NAME_TAP_COUPLER : STRING := 'TapCoupler';
	
	FLEXO_AI_PISTON_LEFT_SENSING_RANGE_MAX : INT := 32767;
	FLEXO_AI_PISTON_LEFT_SENSING_RANGE_MIN : INT := 32767 / 10;
	
	PSD_NUMBER_INTERLOCK_PANELS : UINT := 4;
	PSD_NUMBER_WAFER_PRESENCE_SENSORS : UINT := 2;
	
	PHOTOLUM_NUMBER_INTERLOCK_PANELS : UINT := 3;
	PHOTOLUM_NUMBER_LIGHT_SOURCE : UINT := 4;
	PHOTOLUM_NUMBER_WAFER_PRESENCE_SENSORS : UINT := 3;	
END_VAR

// ---- Shared/GlobalVariables/GlobalConfig.TcGVL
{attribute 'qualified_only'}
VAR_GLOBAL
	AppConfig : AppConfig;
END_VAR

// ---- Shared/GlobalVariables/HardwareGlobalVariables.TcGVL
{attribute 'qualified_only'}
VAR_GLOBAL

	// AttenuationFilter	
	RxBufferAttenuation : ComBuffer;	(* Receive data buffer; used with all receive function blocks *)
	TxBufferAttenuation : ComBuffer;	(* Transmit data buffer; used with all receive function blocks *)	
	
	// PolarisationFilter	
	RxBufferPolarisation : ComBuffer;	(* Receive data buffer; used with all receive function blocks *)
	TxBufferPolarisation : ComBuffer;	(* Transmit data buffer; used with all receive function blocks *)	
	
	// SliderAttenuationFilter	
	RxBufferSliderAttenuation : ComBuffer;	(* Receive data buffer; used with all receive function blocks *)
	TxBufferSliderAttenuation : ComBuffer;	(* Transmit data buffer; used with all receive function blocks *)	
	
	// RotatingSwitch	
	RxBufferRotatingSwitch : ComBuffer;	(* Receive data buffer; used with all receive function blocks *)
	TxBufferRotatingSwitch : ComBuffer;	(* Transmit data buffer; used with all receive function blocks *)	
	
	// SMD12Laser	
	RxBufferLaser : ComBuffer;	(* Receive data buffer; used with all receive function blocks *)
	TxBufferLaser : ComBuffer;	(* Transmit data buffer; used with all receive function blocks *)
	
	// EOLFiberSwitch	
	RxBufferFiberSwitch : ComBuffer;	(* Receive data buffer; used with all receive function blocks *)
	TxBufferFiberSwitch : ComBuffer;	(* Transmit data buffer; used with all receive function blocks *)
	
	// PM101OpticalPowermeter	
	RxBufferOpticalPowermeterHs : ComBuffer;	(* Receive data buffer; used with all receive function blocks *)
	TxBufferOpticalPowermeterHs : ComBuffer;	(* Transmit data buffer; used with all receive function blocks *)
	
	RxBufferOpticalPowermeterHt : ComBuffer;	(* Receive data buffer; used with all receive function blocks *)
	TxBufferOpticalPowermeterHt : ComBuffer;	(* Transmit data buffer; used with all receive function blocks *)
	
	// C13366Mppc	
	RxBufferMppcWide : ComBuffer;	(* Receive data buffer; used with all receive function blocks *)
	TxBufferMppcWide : ComBuffer;	(* Transmit data buffer; used with all receive function blocks *)

	RxBufferMppcNarrow : ComBuffer;	(* Receive data buffer; used with all receive function blocks *)
	TxBufferMppcNarrow : ComBuffer;	(* Transmit data buffer; used with all receive function blocks *)		
	
	// DM430GNScreen	
	RxBufferDM430GNScreenFS : ComBuffer;	(* Receive data buffer; used with all receive function blocks *)
	TxBufferDM430GNScreenFS : ComBuffer;	(* Transmit data buffer; used with all receive function blocks *)
	
	RxBufferDM430GNScreenBS : ComBuffer;	(* Receive data buffer; used with all receive function blocks *)
	TxBufferDM430GNScreenBS : ComBuffer;	(* Transmit data buffer; used with all receive function blocks *)
	
	// FilterWheel	
	RxBufferFilterWheel : ComBuffer;	(* Receive data buffer; used with all receive function blocks *)
	TxBufferFilterWheel : ComBuffer;	(* Transmit data buffer; used with all receive function blocks *)	
	
	// Light
	RxBufferLight : ComBuffer;	(* Receive data buffer; used with all receive function blocks *)
	TxBufferLight : ComBuffer;	(* Transmit data buffer; used with all receive function blocks *)
	
	CyclingCounterReachSetpoint : BOOL;
	
	PwmGenerator : PwmGenerator;
	
	LightState : TExecutionState;
	ChamberState : TExecutionState;
	ChuckState : TExecutionState;
	IonizerState : TExecutionState;
END_VAR

// ---- PMShared/Hardware/Interface/IDevice.TcIO
INTERFACE IDevice

PROPERTY DeviceID : STRING
GET
END_GET
SET
END_SET
END_PROPERTY

PROPERTY Family : DeviceFamily
GET
END_GET
SET
END_SET
END_PROPERTY

PROPERTY Name : STRING
GET
END_GET
SET
END_SET
END_PROPERTY

END_INTERFACE

// ---- PMShared/Hardware/Interface/TrackExecution/IExecution.TcIO
INTERFACE IExecution

PROPERTY Aborted : BOOL
GET
END_GET
SET
END_SET
END_PROPERTY

PROPERTY Busy : BOOL
GET
END_GET
SET
END_SET
END_PROPERTY

PROPERTY Done : BOOL
GET
END_GET
SET
END_SET
END_PROPERTY

PROPERTY Error : BOOL
GET
END_GET
SET
END_SET
END_PROPERTY

PROPERTY ErrorId : UDINT
GET
END_GET
SET
END_SET
END_PROPERTY

PROPERTY Ready : BOOL
GET
END_GET
SET
END_SET
END_PROPERTY

METHOD SetReady
VAR_INPUT
END_VAR
END_METHOD

METHOD Start : BOOL
VAR_INPUT
END_VAR
END_METHOD

END_INTERFACE

// ---- Shared/Log/ILogger.TcIO
INTERFACE ILogger

METHOD Debug
VAR_INPUT
	message : STRING;
END_VAR
END_METHOD

METHOD Error
VAR_INPUT
	message : STRING;
END_VAR
END_METHOD

METHOD Fatal
VAR_INPUT
	message : STRING;
END_VAR
END_METHOD

METHOD Information
VAR_INPUT
	message : STRING;
END_VAR
END_METHOD

METHOD Verbose
VAR_INPUT
	message : STRING;
END_VAR
END_METHOD

METHOD Warning
VAR_INPUT
	message : STRING;
END_VAR
END_METHOD

END_INTERFACE

// ---- Shared/Tools/StringBuilder/ILimitedStringBuilder.TcIO
INTERFACE ILimitedStringBuilder

METHOD Append : IStringBuilder
VAR_INPUT
	text : STRING; 
END_VAR
END_METHOD

METHOD Reset : ILimitedStringBuilder
VAR_INPUT
END_VAR
END_METHOD

METHOD ToString : STRING
VAR_INPUT
END_VAR
END_METHOD

END_INTERFACE

// ---- Shared/Tools/StringBuilder/IStringBuilder.TcIO
INTERFACE IStringBuilder

METHOD Append : IStringBuilder
VAR_INPUT
	text : STRING;
END_VAR
END_METHOD

METHOD InsertAtLocation : REFERENCE TO StringBuilder
VAR_INPUT
	Text : STRING;
    Position : INT;
END_VAR
END_METHOD

METHOD Reset : ILimitedStringBuilder
VAR_INPUT
END_VAR
END_METHOD

METHOD ToString : STRING
VAR_INPUT
END_VAR
END_METHOD

END_INTERFACE

// ---- MAIN.TcPOU
PROGRAM MAIN
VAR	
	HardwareControl : HardwareControl;
END_VAR


HardwareControl();

END_PROGRAM

// ---- Service/HardwareControl.TcPOU
(*
Récupère la Config de AppConfig
Démarre HardwareManager
Todo : Démarre la Bdd
Todo : Démarre le monitoring
*)

FUNCTION_BLOCK HardwareControl
VAR_INPUT
END_VAR
VAR_OUTPUT
END_VAR
VAR
	{region "manage file" }	
	{attribute 'OPC.UA.DA' := '0'}	
	_xml : TXml;	
	{attribute 'hide'}
	_filePath : T_MaxString := Const.APP_CONFIG_FILE_PATH; 
	{attribute 'hide'}  			
    _xPath : T_MaxString := Const.APP_CONFIG_XPATH; 
	{endregion}		
		
	{attribute 'hide'}  
	_loadConfigDone : BOOL;
	{attribute 'OPC.UA.DA' := '0'}
	_initialized : BOOL;
	{attribute 'OPC.UA.DA' := '0'}
	_initializedError : BOOL;	
	{attribute 'OPC.UA.DA' := '0'}
	_message : StringBuilder;
	{attribute 'OPC.UA.DA' := '0'}
	_logger : Logger;
	
	autoBoot : BOOL := TRUE;
	
	HardwareManager : HardwareManager;	
END_VAR

IF autoBoot THEN
	InitHardware();
END_IF

ACTION AppDeserialize:
_xml(FilePath := _filePath, XPath := _xPath, 
	 AddHeaderNodeXml := ADR(GlobalConfig.AppConfig), 
	 SizeOfHeaderNodeXml := SIZEOF(GlobalConfig.AppConfig));
END_ACTION

METHOD PRIVATE InitHardware
VAR_INPUT
END_VAR
VAR	
END_VAR
IF _xml.DeserialisationOperation.Ready AND 
   NOT _initialized THEN
    _logger.Information('Initializing hardware...');
END_IF;

IF NOT _initialized  AND NOT _xml.DeserialisationOperation.Error THEN    
	_xml.DeserialisationOperation.Start();
	AppDeserialize();	
END_IF
 
IF _xml.DeserialisationOperation.Done THEN				
	_logger.Debug(_message.Reset().Append('App configuration from ').
						           Append(TO_STRING(Const.APP_CONFIG_FILE_PATH)).ToString());
		
	_logger.Information('App configuration loading done');				
	_xml.DeserialisationOperation.SetReady();
	
	LoadConfigDone := TRUE;	
	_initialized := TRUE;
END_IF
 
IF NOT _initializedError AND _xml.DeserialisationOperation.Error THEN		
	_logger.Error('App configuration loading error');    		
	_xml.SetError(_xml.DeserialisationOperation.ErrorId);
	
	_initializedError := TRUE;
END_IF

IF _loadConfigDone THEN
	HardwareManager();	
END_IF
END_METHOD

PROPERTY LoadConfigDone : BOOL
GET
LoadConfigDone := _loadConfigDone;
END_GET
SET
_loadConfigDone := LoadConfigDone;
END_SET
END_PROPERTY

END_FUNCTION_BLOCK

// ---- Shared/Tools/Xml/TXml.TcPOU
FUNCTION_BLOCK TXml EXTENDS TExecution
VAR_INPUT
	FilePath : T_MaxString;
	XPath 	 : T_MaxString;
	AddHeaderNodeXml : PVOID;
	SizeOfHeaderNodeXml : UDINT;
END_VAR
VAR_OUTPUT	
END_VAR
VAR
	{attribute 'hide'}		  
	{attribute 'OPC.UA.DA' := '0'}
	_xmlSrvRead : FB_XmlSrvRead;			
	{attribute 'OPC.UA.DA' := '0'}
	_deserialisationOperation : TExecution;	
	{attribute 'OPC.UA.DA' := '0'}
	item : INT;
	{attribute 'OPC.UA.DA' := '0'}
	_logger : Logger;
	{attribute 'OPC.UA.DA' := '0'}
	_message : StringBuilder;
END_VAR

Deserialize(_deserialisationOperation.Starting);

IF _xmlSrvRead.bBusy THEN
    _deserialisationOperation.SetBusy();
END_IF

IF _xmlSrvRead.bError THEN
	_deserialisationOperation.SetError(ErrorId := _xmlSrvRead.nErrId);
		
	_logger.Error(_message.Reset().Append('Xml deserialization - ErrorId : ').
			 			   		   Append(UDINT_TO_STRING(_xmlSrvRead.nErrId)).ToString());
END_IF 

IF _deserialisationOperation.Busy THEN
    IF NOT _xmlSrvRead.bBusy THEN        
        IF THIS^.Aborted THEN
            _deserialisationOperation.SetAborted();
			_logger.Information(_message.Reset().Append('Xml deserialization aborted').ToString());
        ELSE
            _deserialisationOperation.SetDone(); 
			_logger.Debug(_message.Reset().Append('Xml deserialization done').ToString());
        END_IF
    END_IF
END_IF

PROPERTY DeserialisationOperation : IExecution
GET
DeserialisationOperation := _deserialisationOperation;
END_GET
END_PROPERTY

METHOD Deserialize
VAR_INPUT
	Execute : BOOL;
END_VAR
CASE item OF
0:
	IF Execute THEN
		THIS^.State := TExecutionState.Busy;
		_logger.Debug(_message.Reset().Append('Xml deserialization busy').ToString());
		item := item + 1;
	END_IF
1:	
	_xmlSrvRead(
	  pSymAddr	:= AddHeaderNodeXml,
	  cbSymSize	:= SizeOfHeaderNodeXml, 
	  sFilePath	:= FilePath,
	  sXPath	:= XPath,
	  bExecute	:= TRUE
	);	
	item := item + 1;	
		
2:  
	_xmlSrvRead(bExecute:= FALSE);
	IF NOT _xmlSrvRead.bBusy AND NOT _xmlSrvRead.bError THEN		
		THIS^.State := TExecutionState.Ready;
		item := 0;
	END_IF	
END_CASE
END_METHOD

END_FUNCTION_BLOCK

// ---- PMShared/Hardware/Interface/TrackExecution/TExecution.TcPOU
FUNCTION_BLOCK TExecution IMPLEMENTS IExecution 
VAR_INPUT
END_VAR
VAR_OUTPUT
END_VAR
VAR
	{attribute 'OPC.UA.DA' := '1'}
	State : TExecutionState := TExecutionState.Unknown;
	{attribute 'OPC.UA.DA' := '0'}
    _done : BOOL;       
	{attribute 'OPC.UA.DA' := '0'}
    _error : BOOL;      
	{attribute 'OPC.UA.DA' := '0'}
	_warning : BOOL;    
	{attribute 'OPC.UA.DA' := '0'}
    _aborted : BOOL;    
	{attribute 'OPC.UA.DA' := '0'}
    _errorId : UDINT;   
END_VAR

PROPERTY Aborted : BOOL
GET
Aborted := _aborted;
END_GET
SET
_aborted := Aborted;
END_SET
END_PROPERTY

PROPERTY Busy : BOOL
GET
Busy := State = TExecutionState.Busy;
END_GET
SET
END_SET
END_PROPERTY

PROPERTY Done : BOOL
GET
Done := _done;
END_GET
SET
_done := Done;
END_SET
END_PROPERTY

PROPERTY Error : BOOL
GET
Error := _error;
END_GET
SET
_error := Error;
END_SET
END_PROPERTY

PROPERTY ErrorId : UDINT
GET
ErrorId := _errorId;
END_GET
SET
_errorId := ErrorId;
END_SET
END_PROPERTY

PROPERTY Ready : BOOL;
GET
Ready := State = TExecutionState.Ready;
END_GET
SET
END_SET
END_PROPERTY

METHOD SetAborted
VAR_INPUT
END_VAR
_aborted := TRUE;
State := TExecutionState.Ready;
END_METHOD

METHOD SetBusy
VAR_INPUT
END_VAR
IF State = TExecutionState.Starting THEN
    State := TExecutionState.Busy;
END_IF
END_METHOD

METHOD SetDone 
VAR_INPUT
END_VAR
_done := TRUE;
State := TExecutionState.Ready;
END_METHOD

METHOD SetError
VAR_INPUT
	ErrorId : UDINT;
END_VAR
_error := TRUE;
_errorId := ErrorId;
State := TExecutionState.Error;
END_METHOD

METHOD SetReady
VAR_INPUT
END_VAR
// Clear results
_done := FALSE;
_error := FALSE;
_errorId := 0;
_aborted := FALSE;

State := TExecutionState.Ready;
END_METHOD

METHOD SetWarning
VAR_INPUT
END_VAR
_warning := TRUE;
State := TExecutionState.Ready;
END_METHOD

METHOD Start : BOOL
VAR_INPUT
END_VAR
IF State = TExecutionState.Ready OR 
    State = TExecutionState.Unknown THEN
    // Acq results
    _done := FALSE;
    _error := FALSE;
    _errorId := 0;
    _aborted := FALSE;
 
    State := TExecutionState.Starting;
 
    Start := TRUE;
END_IF
END_METHOD

PROPERTY Starting : BOOL
GET
Starting := State = TExecutionState.Starting ;
END_GET
SET
END_SET
END_PROPERTY

PROPERTY Status : TExecutionState
GET
Status := State;
END_GET
SET
State := Status;
END_SET
END_PROPERTY

PROPERTY Warning : BOOL
GET
Warning := _warning;
END_GET
SET
_warning := Warning;
END_SET
END_PROPERTY

END_FUNCTION_BLOCK

// ---- Shared/Log/Logger.TcPOU
FUNCTION_BLOCK Logger IMPLEMENTS ILogger
VAR_INPUT
END_VAR
VAR_OUTPUT
	ipResultMessage : I_TcMessage := fbResult;
END_VAR
VAR
	fbResult : FB_TcMessage;
	fbSource : FB_TcSourceInfo;
	
	hrLastInternalError : HRESULT;	
END_VAR

METHOD Debug
VAR_INPUT
	message	: STRING;
END_VAR
VAR
	hr : HRESULT;
END_VAR
hr := fbResult.CreateEx(TC_EVENTS.EventLoggerPlc.PlcEventDebug, ipSourceInfo:=fbSource);
Write(message, hr);
END_METHOD

METHOD Error
VAR_INPUT
	message	: STRING;
END_VAR
VAR
	hr : HRESULT;
END_VAR
hr := fbResult.CreateEx(TC_EVENTS.EventLoggerPlc.PlcEventError, ipSourceInfo:=fbSource);
Write(message, hr);
END_METHOD

METHOD Fatal
VAR_INPUT
	message	: STRING;
END_VAR
VAR
	hr : HRESULT;
END_VAR
hr := fbResult.CreateEx(TC_EVENTS.EventLoggerPlc.PlcEventFatal, ipSourceInfo:=fbSource);
Write(message, hr);
END_METHOD

METHOD Information
VAR_INPUT
	message	: STRING;
END_VAR
VAR
	hr : HRESULT;
END_VAR
hr := fbResult.CreateEx(TC_EVENTS.EventLoggerPlc.PlcEventInformation, ipSourceInfo:=fbSource);
Write(message, hr);
END_METHOD

METHOD Verbose
VAR_INPUT
	message	: STRING;
END_VAR
VAR
	hr : HRESULT;
END_VAR
hr := fbResult.CreateEx(TC_EVENTS.EventLoggerPlc.PlcEventVerbose, ipSourceInfo:=fbSource);
Write(message, hr);
END_METHOD

METHOD Warning
VAR_INPUT
	message	: STRING;
END_VAR
VAR
	hr : HRESULT;
END_VAR
hr := fbResult.CreateEx(TC_EVENTS.EventLoggerPlc.PlcEventWarning, ipSourceInfo:=fbSource);
Write(message, hr);
END_METHOD

METHOD PRIVATE Write
VAR_INPUT
	message : STRING;
	handle : HRESULT;
END_VAR
fbResult.ipArguments.Clear().AddString(message);

IF fbResult.eSeverity >= TcEventSeverity.Verbose THEN
	handle := fbResult.Send(0);
	IF FAILED(handle) THEN
		hrLastInternalError := handle;
	END_IF
END_IF
END_METHOD

END_FUNCTION_BLOCK

// ---- Shared/Tools/StringBuilder/StringBuilder.TcPOU
FUNCTION_BLOCK StringBuilder IMPLEMENTS IStringBuilder, ILimitedStringBuilder
VAR_INPUT
END_VAR
VAR_OUTPUT
END_VAR
VAR
	{attribute 'hide'}
    _workString : STRING;
END_VAR

METHOD Append : IStringBuilder
VAR_INPUT
    text : STRING; 
END_VAR
_workString := CONCAT(_workString, text);
Append := THIS^;
END_METHOD

METHOD InsertAtLocation : REFERENCE TO StringBuilder
VAR_INPUT
    Text : STRING;
    Position : INT;
END_VAR
_workString := Tc2_Standard.INSERT(_WorkString, Text, Position);
InsertAtLocation REF= THIS^;
END_METHOD

METHOD Reset : ILimitedStringBuilder
_workString := '';
Reset := THIS^;
END_METHOD

METHOD ToString : STRING
ToString := _workString;
END_METHOD

END_FUNCTION_BLOCK

// ---- PMShared/Hardware/Common/HardwareManager.TcPOU
(* Initialise les devices *)
FUNCTION_BLOCK HardwareManager
VAR_INPUT			
END_VAR
VAR_OUTPUT
END_VAR
VAR	
	{attribute 'OPC.UA.DA' := '0'}
	{attribute 'OPC.UA.DA.StructuredType' := '0'}
	ProcessModulesConfig : ProcessModulesConfig;	

	{attribute 'OPC.UA.DA' := '0'}
	{attribute 'OPC.UA.DA.StructuredType' := '0'}
	CalibratePMsConfig : CalibratePMsConfig;
	
	{region "PMs" } 	
	
	{attribute 'OPC.UA.DA' := '1'}
	{attribute 'OPC.UA.DA.StructuredType' := '1'}	 
	Lightspeed : Lightspeed(Config := ProcessModulesConfig.LightspeedConfig, CalibrateConfig := CalibratePMsConfig.LsCalibrateConfig);

	{attribute 'OPC.UA.DA' := '1'}
	{attribute 'OPC.UA.DA.StructuredType' := '1'}			
	Psd : Psd(Config := ProcessModulesConfig.PsdConfig);
		
	{attribute 'OPC.UA.DA' := '1'}
	{attribute 'OPC.UA.DA.StructuredType' := '1'}	 
	Nst : Nst(Config := ProcessModulesConfig.NstConfig);
 
	{attribute 'OPC.UA.DA' := '1'}
	{attribute 'OPC.UA.DA.StructuredType' := '1'}	 
	PhotoLum : PhotoLum(Config := ProcessModulesConfig.PhotoLumConfig);
		   
	{endregion}
					  	
	{attribute 'hide'}  
	_initializedHardware : BOOL;
	{attribute 'hide'}  
	_initializedCalibrate : BOOL ; //:= TRUE;  TODO pourquoi la calibration de la NST pose problème ? 
	
	{attribute 'OPC.UA.DA' := '0'}
	_xmlCalibrate : TXml;
	{attribute 'OPC.UA.DA' := '0'}
	_xmlHardware : TXml;
	{attribute 'OPC.UA.DA' := '0'}
	_logger : Logger;
	{attribute 'OPC.UA.DA' := '0'}
	_message : StringBuilder;
		
END_VAR

IF NOT _initializedCalibrate AND NOT _xmlCalibrate.DeserialisationOperation.Error THEN  
	InitCalibrate();	
END_IF	

IF _initializedCalibrate AND NOT _initializedHardware AND NOT 
	_xmlHardware.DeserialisationOperation.Error THEN
	
	InitHardware();
END_IF

IF  _initializedHardware AND _initializedCalibrate THEN
	IF ProcessModulesConfig.LightspeedConfig.IsEnabled THEN
		Lightspeed();	
	END_IF

	IF ProcessModulesConfig.PsdConfig.IsEnabled THEN
		Psd();	
	END_IF		
	
	IF ProcessModulesConfig.NstConfig.IsEnabled THEN
		Nst();	
	END_IF
	
	IF ProcessModulesConfig.PhotoLumConfig.IsEnabled THEN
		PhotoLum();	
	END_IF
END_IF

ACTION CalibrateDeserialize:
_xmlCalibrate(FilePath := GlobalConfig.AppConfig.CalibrateConfig.CalibratePath, 
	 		  XPath := GlobalConfig.AppConfig.CalibrateConfig.CalibrateHeaderNodeXml,  
	 		  AddHeaderNodeXml := ADR(CalibratePMsConfig), 
	 		  SizeOfHeaderNodeXml := SIZEOF(CalibratePMsConfig));
END_ACTION

ACTION HardwareDeserialize:
_xmlHardware(FilePath := GlobalConfig.AppConfig.LogConfig.LogFileConfigPath, 
	 		 XPath := GlobalConfig.AppConfig.LogConfig.HeaderNodeXml, 
	 		 AddHeaderNodeXml := ADR(ProcessModulesConfig), 
	 		 SizeOfHeaderNodeXml := SIZEOF(ProcessModulesConfig));
END_ACTION

METHOD InitCalibrate : BOOL
VAR_INPUT
END_VAR

IF _xmlCalibrate.DeserialisationOperation.Ready THEN
	_logger.Information(_message.Reset().Append('Loading calibrate configuration from ').
						    		 	 Append(TO_STRING(GlobalConfig.AppConfig.CalibrateConfig.CalibratePath)).ToString());
END_IF;	

_xmlCalibrate.DeserialisationOperation.Start();
CalibrateDeserialize();
	
IF _xmlCalibrate.DeserialisationOperation.Done THEN
	_logger.Information('Calibrate configuration loading done');	
	_xmlCalibrate.DeserialisationOperation.SetReady();		
	
	_initializedCalibrate := TRUE;
END_IF
 
IF _xmlCalibrate.DeserialisationOperation.Error THEN	
	_logger.Error('Calibrate load initialization error '); 
	_xmlCalibrate.SetError(_xmlCalibrate.DeserialisationOperation.ErrorId);
	
	_initializedCalibrate := FALSE;
END_IF
END_METHOD

METHOD PRIVATE InitHardware : BOOL
VAR_INPUT
END_VAR
VAR
END_VAR

IF _xmlHardware.DeserialisationOperation.Ready THEN
	_logger.Information(_message.Reset().Append('Loading hardware configuration from ').
						    		 	 Append(TO_STRING(GlobalConfig.AppConfig.LogConfig.LogFileConfigPath)).ToString());
END_IF;	

_xmlHardware.DeserialisationOperation.Start();
HardwareDeserialize();
	
IF _xmlHardware.DeserialisationOperation.Done THEN
	_logger.Information('Hardware configuration loading done');	
	_xmlHardware.DeserialisationOperation.SetReady();	
	
	// Load PMs
	IF ProcessModulesConfig.LightspeedConfig.IsEnabled THEN
		InitializeLightspeed();	
	END_IF
	
	IF ProcessModulesConfig.PsdConfig.IsEnabled THEN
		InitializePsd();	
	END_IF
	
	IF ProcessModulesConfig.NstConfig.IsEnabled THEN
		InitializeNst();	
	END_IF
	
	IF ProcessModulesConfig.PhotoLumConfig.IsEnabled THEN
		InitializePhotoLum();	
	END_IF
	
	_initializedHardware := TRUE;
END_IF
 
IF _xmlHardware.DeserialisationOperation.Error THEN	
	_logger.Error('Hardware load initialization error'); 
	_xmlHardware.SetError(_xmlHardware.DeserialisationOperation.ErrorId);
	
	_initializedHardware := FALSE;
END_IF
END_METHOD

METHOD InitializeLightspeed 
VAR_INPUT
END_VAR
Lightspeed.FB_init(FALSE, FALSE, Config := ProcessModulesConfig.LightspeedConfig, CalibrateConfig := CalibratePMsConfig.LsCalibrateConfig);
END_METHOD

METHOD InitializeNst 
VAR_INPUT
END_VAR
Nst.FB_init(FALSE, FALSE, Config := ProcessModulesConfig.NstConfig);
END_METHOD

METHOD InitializePhotoLum 
VAR_INPUT
END_VAR
PhotoLum.FB_init(FALSE, FALSE, Config := ProcessModulesConfig.PhotoLumConfig);
END_METHOD

METHOD InitializePsd 
VAR_INPUT
END_VAR
Psd.FB_init(FALSE, FALSE, Config := ProcessModulesConfig.PsdConfig);
END_METHOD

END_FUNCTION_BLOCK

// ---- Service/PMs/Lightspeed/Lightspeed.TcPOU
FUNCTION_BLOCK Lightspeed EXTENDS PlcModule
VAR_INPUT
	
	{attribute 'OPC.UA.DA' := '0'}
	LightspeedConfig : LightspeedConfig;
	
	{attribute 'OPC.UA.DA' := '0'}
	LsCalibrateConfig : LsCalibrateConfig;
	
	(* Chamber *)
	Chamber : LightspeedChamber(Config := LightspeedConfig.ChamberConfigs.LightspeedChamberConfig);
		
	(* AttenuationFilterConfigs *) 
	FW212CAttenuationFilter : FW212CAttenuationFilter(Config := LightspeedConfig.AttenuationFilterConfigs.FW212CAttenuationFilterConfig);
	ELL14KAttenuationFilter : ELL14KAttenuationFilter(Config := LightspeedConfig.AttenuationFilterConfigs.ELL14KAttenuationFilterConfig);
	ELL9AttenuationFilter : ELL9AttenuationFilter(Config := LightspeedConfig.AttenuationFilterConfigs.ELL9AttenuationFilterConfig);
	
	(* Slider Attenuation *)
	ELL6SliderAttenuationFilter : ELL6AttenuationFilter(Config := LightspeedConfig.SliderAttenuationFilterConfigs.ELL6SliderFilterConfig);													
	
	(* Rotating switch *) 
	ELL18RotatingSwitch : ELL18AttenuationFilter(Config := LightspeedConfig.RotatingSwitchConfigs.ELL18RotatingSwitchConfig);
	
	(* PolarisationFilterConfigs *) 
	FW212CPolarisationFilter : FW212CPolarisationFilter(Config := LightspeedConfig.PolarisationFilterConfigs.FW212CPolarisationFilterConfig);
	ELL14KPolarisationFilter : ELL14KPolarisationFilter(Config := LightspeedConfig.PolarisationFilterConfigs.ELL14KPolarisationFilterConfig, 
														HsPolarisationConfig := LsCalibrateConfig.HSPowermeter.PolarisationConfig,
														HtPolarisationConfig := LsCalibrateConfig.HTPowermeter.PolarisationConfig);
		
	
	(* LaserConfigs *) 
	SMD12Laser : SMD12Laser(Config := LightspeedConfig.LaserConfigs.SMD12LaserConfig);
	Sapphire488Laser : Sapphire488Laser(Config := LightspeedConfig.LaserConfigs.Sapphire488LaserConfig);
	
	(* FiberSwitchConfigs *) 
	EOLFiberSwitch : EOLFiberSwitch(Config := LightspeedConfig.FiberSwitchConfigs.EOLFiberSwitchConfig);
	
	(* OpticalPowermeterConfigs *) 
	PM101OpticalPowermeterHs : PM101OpticalPowermeterHs(Config := LightspeedConfig.OpticalPowermeterConfigs.PM101OpticalPowermeterConfigHs, 
														PolarisationConfig := LsCalibrateConfig.HSPowermeter.PolarisationConfig,
														RFactorSettings := LsCalibrateConfig.HSPowermeter.RFactorSettings,
														ResponsivityConfig := LsCalibrateConfig.HSPowermeter.ResponsivityConfig);
	PM101OpticalPowermeterHt : PM101OpticalPowermeterHt(Config := LightspeedConfig.OpticalPowermeterConfigs.PM101OpticalPowermeterConfigHt, 
														PolarisationConfig := LsCalibrateConfig.HTPowermeter.PolarisationConfig, 
														RFactorSettings := LsCalibrateConfig.HTPowermeter.RFactorSettings,
														ResponsivityConfig := LsCalibrateConfig.HTPowermeter.ResponsivityConfig);
	
	(* DistanceSensorConfigs *) 
	MicroEpsilonDistanceSensor : MicroEpsilonDistanceSensor(Config := LightspeedConfig.DistanceSensorConfigs.MicroEpsilonDistanceSensorConfig);
	
	(* MppcConfigs *) 
	C13336MppcWide   : C13336MppcWide(Config := LightspeedConfig.MppcConfigs.C13336MppcConfigWide);
	C13336MppcNarrow : C13366MppcNarrow(Config := LightspeedConfig.MppcConfigs.C13336MppcConfigNarrow);
	
	(* ShutterConfigs *)
	Ed12dssShutter : Ed12dssShutter(Config := LightspeedConfig.ShutterConfigs.Ed12dssShutterConfig);
	Sh10pilShutter : Sh10pilShutter(Config := LightspeedConfig.ShutterConfigs.Sh10pilShutterConfig);
	
	(* FastAttenuationConfigs *)
	Std900FastAttenuation : Std900FastAttenuation(Config := LightspeedConfig.FastAttenuationConfigs.Std900FastAttenuationConfig);	
	
END_VAR
VAR_OUTPUT
END_VAR
VAR
	{attribute 'OPC.UA.DA' := '0'}
	_startCycling : BOOL;
	{attribute 'OPC.UA.DA' := '0'}
	_count : UINT;
	{attribute 'OPC.UA.DA' := '0'}
	_ActivateCyclingMotorOpen : BOOL ; (* 0 = close door ; 1 = open door  *) 
	{attribute 'OPC.UA.DA' := '0'}
	_CyclingCounterReachSetpoint : BOOL ;
	{attribute 'OPC.UA.DA' := '0'}
	OpenCloseCyclingCount : WORD := 10; (* default value *) 
	{attribute 'OPC.UA.DA' := '0'}
	OpenCloseCurrentCounterValue : WORD:= 0; (* init value *)  ;
	{attribute 'OPC.UA.DA' := '0'}
	WaitingTimer : TON;
	{attribute 'OPC.UA.DA' := '0'}
	DoorSlitOpenCloseCounter: CTU;
	{attribute 'OPC.UA.DA' := '0'}
	OpenCloseCyclingCounterReset : BOOL := FALSE; 
	{attribute 'OPC.UA.DA' := '0'}
	_stopCycling: BOOL:= FALSE;	
	
	{attribute 'OPC.UA.DA' := '0'}
	_mppcActivate : BOOL := TRUE; //TODO à remettre 
	
END_VAR


SUPER^();

IF LightspeedConfig.ChamberConfigs.LightspeedChamberConfig.IsEnabled THEN
	Chamber(MppcActivate => _mppcActivate);	
	
	Door_Slit_Ctrl();
	OpenCloseCycling(_startCycling, _count);
	StopCycling(_stopCycling);	
END_IF

(* Attenuation *)
IF LightspeedConfig.AttenuationFilterConfigs.FW212CAttenuationFilterConfig.IsEnabled THEN		
	FW212CAttenuationFilter();
	IF FW212CAttenuationFilter.InitConfigSerialCom THEN
		;
	END_IF
ELSIF LightspeedConfig.AttenuationFilterConfigs.ELL14KAttenuationFilterConfig.IsEnabled THEN		
	ELL14KAttenuationFilter();
	IF ELL14KAttenuationFilter.InitConfigSerialCom THEN
		;
	END_IF
ELSIF LightspeedConfig.AttenuationFilterConfigs.ELL9AttenuationFilterConfig.IsEnabled THEN		
	ELL9AttenuationFilter();
	IF ELL9AttenuationFilter.InitConfigSerialCom THEN
		;
	END_IF		
END_IF

(* Slider Attenuation *)
IF LightspeedConfig.Version = '2' THEN
	IF LightspeedConfig.SliderAttenuationFilterConfigs.ELL6SliderFilterConfig.IsEnabled THEN		
		ELL6SliderAttenuationFilter();
		IF ELL6SliderAttenuationFilter.InitConfigSerialCom THEN
			;
		END_IF
	END_IF
END_IF

(* Rotating switch *)
IF LightspeedConfig.Version = '2' THEN
	IF LightspeedConfig.RotatingSwitchConfigs.ELL18RotatingSwitchConfig.IsEnabled THEN		
		ELL18RotatingSwitch();
		IF ELL18RotatingSwitch.InitConfigSerialCom THEN
			;
		END_IF
	END_IF
END_IF

IF LightspeedConfig.PolarisationFilterConfigs.FW212CPolarisationFilterConfig.IsEnabled THEN
	FW212CPolarisationFilter();	
	IF FW212CPolarisationFilter.InitConfigSerialCom THEN
		;
	END_IF
ELSIF LightspeedConfig.PolarisationFilterConfigs.ELL14KPolarisationFilterConfig.IsEnabled THEN		
	ELL14KPolarisationFilter();
	IF ELL14KPolarisationFilter.InitConfigSerialCom THEN
		;
	END_IF			
END_IF

IF LightspeedConfig.LaserConfigs.SMD12LaserConfig.IsEnabled THEN
	SMD12Laser();
	IF SMD12Laser.InitConfigSerialCom THEN
		;
	END_IF
ELSIF LightspeedConfig.LaserConfigs.Sapphire488LaserConfig.IsEnabled THEN
	Sapphire488Laser();
	IF Sapphire488Laser.InitConfigSerialCom THEN
		;
	END_IF
ELSIF LightspeedConfig.LaserConfigs.Sapphire488LaserConfig.IsEnabled THEN
	Sapphire488Laser();
	IF Sapphire488Laser.InitConfigSerialCom THEN
		;
	END_IF	
END_IF

IF LightspeedConfig.FiberSwitchConfigs.EOLFiberSwitchConfig.IsEnabled THEN
	EOLFiberSwitch();
	IF EOLFiberSwitch.InitConfigSerialCom THEN
		;
	END_IF
END_IF

IF LightspeedConfig.OpticalPowermeterConfigs.PM101OpticalPowermeterConfigHs.IsEnabled OR 
   LightspeedConfig.OpticalPowermeterConfigs.PM101OpticalPowermeterConfigHs.IsSimulated THEN
	PM101OpticalPowermeterHs(PolarResult := ELL14KPolarisationFilter.PolarResult);
	IF PM101OpticalPowermeterHs.InitConfigSerialCom THEN
		;
	END_IF	
END_IF

IF LightspeedConfig.OpticalPowermeterConfigs.PM101OpticalPowermeterConfigHt.IsEnabled THEN
	PM101OpticalPowermeterHt(PolarResult := ELL14KPolarisationFilter.PolarResult);
	IF PM101OpticalPowermeterHt.InitConfigSerialCom THEN
		;
	END_IF	
END_IF

IF LightspeedConfig.DistanceSensorConfigs.MicroEpsilonDistanceSensorConfig.IsEnabled THEN
	MicroEpsilonDistanceSensor();	
END_IF

IF LightspeedConfig.MppcConfigs.C13336MppcConfigWide.IsEnabled THEN
	C13336MppcWide(MppcActivate := _mppcActivate);
	IF C13336MppcWide.InitConfigSerialCom THEN
		;
	END_IF
END_IF

IF LightspeedConfig.MppcConfigs.C13336MppcConfigNarrow.IsEnabled THEN
	C13336MppcNarrow(MppcActivate := _mppcActivate);
	IF C13336MppcNarrow.InitConfigSerialCom THEN
		;
	END_IF
END_IF

IF LightspeedConfig.ShutterConfigs.Ed12dssShutterConfig.IsEnabled THEN
	Ed12dssShutter();	
ELSIF LightspeedConfig.ShutterConfigs.SH10PILShutterConfig.IsEnabled THEN
	Sh10pilShutter();
END_IF

IF LightspeedConfig.FastAttenuationConfigs.Std900FastAttenuationConfig.IsEnabled THEN
	Std900FastAttenuation();	
END_IF

METHOD Door_Slit_Ctrl : BOOL
VAR_INPUT	
END_VAR
VAR
	timeout : TIME := T#1400MS; (* 2 * open time (700ms)  *) 
	MotorTurnOffAfterTimeout: TON;
END_VAR
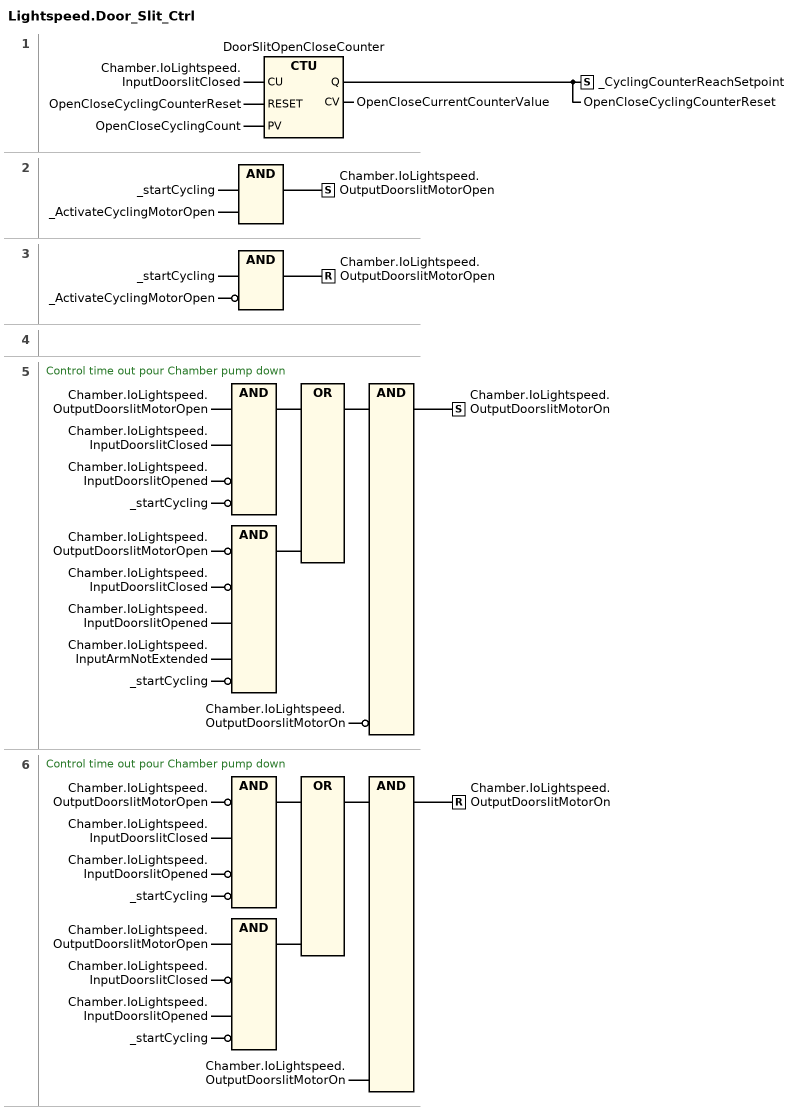
// NETWORK 1
DoorSlitOpenCloseCounter(
    CU := Chamber.IoLightspeed.InputDoorslitClosed,
    RESET := OpenCloseCyclingCounterReset,
    PV := OpenCloseCyclingCount,
    CV => OpenCloseCurrentCounterValue); // CTU
_CyclingCounterReachSetpoint S= DoorSlitOpenCloseCounter.Q;
OpenCloseCyclingCounterReset := DoorSlitOpenCloseCounter.Q;

// NETWORK 2
Chamber.IoLightspeed.OutputDoorslitMotorOpen S= _startCycling AND _ActivateCyclingMotorOpen;

// NETWORK 3
Chamber.IoLightspeed.OutputDoorslitMotorOpen R= _startCycling AND NOT _ActivateCyclingMotorOpen;

// NETWORK 4

// NETWORK 5
// Control time out pour Chamber pump down
Chamber.IoLightspeed.OutputDoorslitMotorOn S= (Chamber.IoLightspeed.OutputDoorslitMotorOpen AND Chamber.IoLightspeed.InputDoorslitClosed AND NOT Chamber.IoLightspeed.InputDoorslitOpened AND NOT _startCycling OR NOT Chamber.IoLightspeed.OutputDoorslitMotorOpen AND NOT Chamber.IoLightspeed.InputDoorslitClosed AND Chamber.IoLightspeed.InputDoorslitOpened AND Chamber.IoLightspeed.InputArmNotExtended AND NOT _startCycling) AND NOT Chamber.IoLightspeed.OutputDoorslitMotorOn;

// NETWORK 6
// Control time out pour Chamber pump down
Chamber.IoLightspeed.OutputDoorslitMotorOn R= (NOT Chamber.IoLightspeed.OutputDoorslitMotorOpen AND Chamber.IoLightspeed.InputDoorslitClosed AND NOT Chamber.IoLightspeed.InputDoorslitOpened AND NOT _startCycling OR Chamber.IoLightspeed.OutputDoorslitMotorOpen AND NOT Chamber.IoLightspeed.InputDoorslitClosed AND Chamber.IoLightspeed.InputDoorslitOpened AND NOT _startCycling) AND Chamber.IoLightspeed.OutputDoorslitMotorOn;

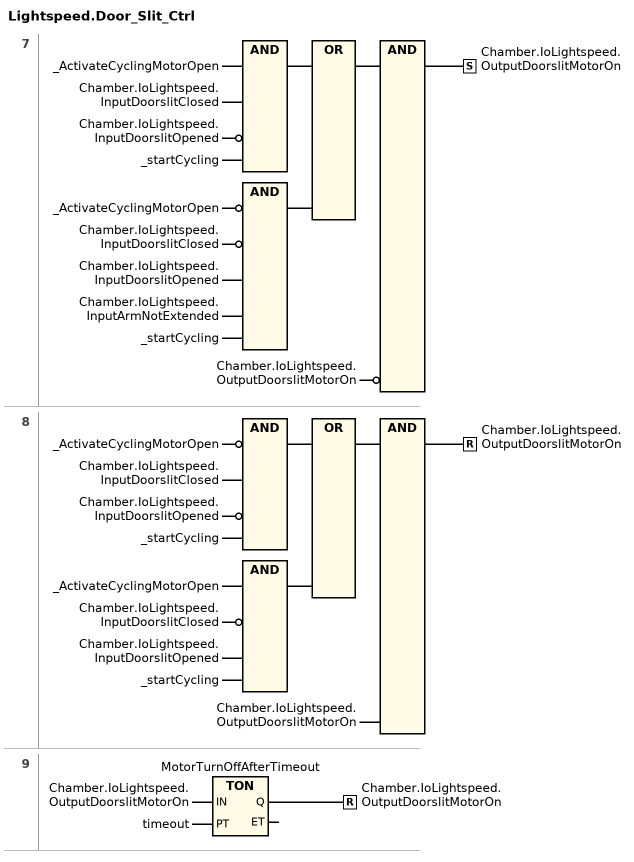
// NETWORK 7
Chamber.IoLightspeed.OutputDoorslitMotorOn S= (_ActivateCyclingMotorOpen AND Chamber.IoLightspeed.InputDoorslitClosed AND NOT Chamber.IoLightspeed.InputDoorslitOpened AND _startCycling OR NOT _ActivateCyclingMotorOpen AND NOT Chamber.IoLightspeed.InputDoorslitClosed AND Chamber.IoLightspeed.InputDoorslitOpened AND Chamber.IoLightspeed.InputArmNotExtended AND _startCycling) AND NOT Chamber.IoLightspeed.OutputDoorslitMotorOn;

// NETWORK 8
Chamber.IoLightspeed.OutputDoorslitMotorOn R= (NOT _ActivateCyclingMotorOpen AND Chamber.IoLightspeed.InputDoorslitClosed AND NOT Chamber.IoLightspeed.InputDoorslitOpened AND _startCycling OR _ActivateCyclingMotorOpen AND NOT Chamber.IoLightspeed.InputDoorslitClosed AND Chamber.IoLightspeed.InputDoorslitOpened AND _startCycling) AND Chamber.IoLightspeed.OutputDoorslitMotorOn;

// NETWORK 9
MotorTurnOffAfterTimeout(IN := Chamber.IoLightspeed.OutputDoorslitMotorOn, PT := timeout); // TON
Chamber.IoLightspeed.OutputDoorslitMotorOn R= MotorTurnOffAfterTimeout.Q;
END_METHOD

METHOD FB_init : BOOL
VAR_INPUT
	bInitRetains : BOOL; // if TRUE, the retain variables are initialized (warm start / cold start)
	bInCopyCode : BOOL;  // if TRUE, the instance afterwards gets moved into the copy code (online change)
	Config : LightspeedConfig;
	CalibrateConfig : LsCalibrateConfig;
END_VAR
LightspeedConfig := Config;
LsCalibrateConfig := CalibrateConfig;
LsBkgrdLsSerialCom(Config := LightspeedConfig);

IF Config.IsEnabled THEN
	_logger.Information('Lightspeed devices initialization starting...');
END_IF	

(* Chamber *)
IF Config.ChamberConfigs.LightspeedChamberConfig.IsEnabled THEN
	Chamber.FB_init(FALSE, FALSE, Config := Config.ChamberConfigs.LightspeedChamberConfig);	
END_IF

(* AttenuationFilterConfigs *)
IF Config.AttenuationFilterConfigs.FW212CAttenuationFilterConfig.IsEnabled THEN
	FW212CAttenuationFilter.FB_init(FALSE, FALSE, Config := Config.AttenuationFilterConfigs.FW212CAttenuationFilterConfig);	
ELSIF Config.AttenuationFilterConfigs.ELL14KAttenuationFilterConfig.IsEnabled THEN
	ELL14KAttenuationFilter.FB_init(FALSE, FALSE, Config := Config.AttenuationFilterConfigs.ELL14KAttenuationFilterConfig);
END_IF

(* Slider Attenuation *)
IF Config.Version = '2' THEN
	IF Config.SliderAttenuationFilterConfigs.ELL6SliderFilterConfig.IsEnabled THEN
		ELL6SliderAttenuationFilter.FB_init(FALSE, FALSE, Config := Config.SliderAttenuationFilterConfigs.ELL6SliderFilterConfig);
	END_IF
END_IF

(* Rotating switch *)
IF Config.Version = '2' THEN
	IF Config.RotatingSwitchConfigs.ELL18RotatingSwitchConfig.IsEnabled THEN
		ELL18RotatingSwitch.FB_init(FALSE, FALSE, Config := Config.RotatingSwitchConfigs.ELL18RotatingSwitchConfig);
	END_IF
END_IF

(* PolarisationFilterConfigs *)
IF Config.PolarisationFilterConfigs.FW212CPolarisationFilterConfig.IsEnabled THEN
	FW212CPolarisationFilter.FB_init(FALSE, FALSE, Config := Config.PolarisationFilterConfigs.FW212CPolarisationFilterConfig);	
ELSIF Config.PolarisationFilterConfigs.ELL14KPolarisationFilterConfig.IsEnabled THEN
	ELL14KPolarisationFilter.FB_init(FALSE, FALSE, Config := Config.PolarisationFilterConfigs.ELL14KPolarisationFilterConfig, 
												   HsPolarisationConfig := CalibrateConfig.HSPowermeter.PolarisationConfig,
												   HtPolarisationConfig := CalibrateConfig.HTPowermeter.PolarisationConfig);
END_IF

(* LaserConfigs *) 
IF Config.LaserConfigs.SMD12LaserConfig.IsEnabled THEN
	SMD12Laser.FB_init(FALSE, FALSE, Config := Config.LaserConfigs.SMD12LaserConfig);	
ELSIF Config.LaserConfigs.Sapphire488LaserConfig.IsEnabled THEN
	Sapphire488Laser.FB_init(FALSE, FALSE, Config := Config.LaserConfigs.Sapphire488LaserConfig);	
END_IF

(* FiberSwitchConfigs *) 
IF Config.FiberSwitchConfigs.EOLFiberSwitchConfig.IsEnabled THEN
	EOLFiberSwitch.FB_init(FALSE, FALSE, Config := Config.FiberSwitchConfigs.EOLFiberSwitchConfig);	
END_IF

